# B&R Automation Studio project BaseProject (part 4)

#### Cyclic.st - Init, cyclic, exit code
```iecst
PROGRAM _CYCLIC

	MC_BR_SegCommandError_AcpTrak_0(Segment := ADR(TrackDiag.Seg.SegList[0].McType));

	IF MC_BR_SegCommandError_AcpTrak_0.Done THEN
		MC_BR_SegCommandError_AcpTrak_0.Execute := FALSE;
	END_IF

	(***********************************ASSEMBLY INFORMATION******************************	)
	(*Read Assebly Status*)

	DiagFbs.Asm.ReadStatus.Enable	:= TRUE;
	DiagFbs.Asm.ReadStatus();

	IF DiagFbs.Asm.ReadStatus.Valid THEN
		TrackDiag.Asm.AssemblyDisabled 	:= DiagFbs.Asm.ReadStatus.AssemblyDisabled;
		TrackDiag.Asm.AssemblyErrorStop := DiagFbs.Asm.ReadStatus.AssemblyErrorStop;
		TrackDiag.Asm.AssemblyReady		:= DiagFbs.Asm.ReadStatus.AssemblyReady;
		TrackDiag.Asm.AssemblyHoming	:= DiagFbs.Asm.ReadStatus.AssemblyHoming;
		TrackDiag.Asm.AssemblyStopping	:= DiagFbs.Asm.ReadStatus.AssemblyStopping;
	END_IF

	(*Read Assembly Info *)

	DiagFbs.Asm.ReadInfo.Enable		:= TRUE;
	DiagFbs.Asm.ReadInfo();

	IF DiagFbs.Asm.ReadInfo.Valid THEN
		TrackDiag.Asm.CommunicationReady 	:= DiagFbs.Asm.ReadInfo.AssemblyInfo.CommunicationReady;
		TrackDiag.Asm.PowerOn				:= DiagFbs.Asm.ReadInfo.AssemblyInfo.PowerOn;
		TrackDiag.Asm.ReadyForPowerOn		:= DiagFbs.Asm.ReadInfo.AssemblyInfo.ReadyForPowerOn;
		TrackDiag.Asm.ShuttleInErrorStopCount := DiagFbs.Asm.ReadInfo.AssemblyInfo.ShuttlesInErrorStopCount;
		TrackDiag.Asm.StartupCount			:= DiagFbs.Asm.ReadInfo.AssemblyInfo.StartupCount;
	END_IF

	(****************************** SEGMENT ERROR INFORMATION *****************************************)

	FOR SegIndex := 0 TO NUM_SEG DO

		IF TrackDiag.Seg.SegList[SegIndex].McType.controlif <> 0 THEN //If the array contains a segment reference

			DiagFbs.Seg.ReadInfo[SegIndex].Segment 	:= ADR(TrackDiag.Seg.SegList[SegIndex].McType);
			DiagFbs.Seg.ReadInfo[SegIndex].Enable	:= TRUE;
			DiagFbs.Seg.ReadInfo[SegIndex]();

			IF DiagFbs.Seg.ReadInfo[SegIndex].Valid THEN
				//Capture Segment Info
				TrackDiag.Seg.SegList[SegIndex].Status.CommunicationReady 	:= DiagFbs.Seg.ReadInfo[SegIndex].SegmentInfo.CommunicationReady;
				TrackDiag.Seg.SegList[SegIndex].Status.ReadyForPowerOn		:= DiagFbs.Seg.ReadInfo[SegIndex].SegmentInfo.ReadyForPowerOn;
				TrackDiag.Seg.SegList[SegIndex].Status.PowerOn				:= DiagFbs.Seg.ReadInfo[SegIndex].SegmentInfo.PowerOn;
				TrackDiag.Seg.SegList[SegIndex].Status.StartupCount			:= DiagFbs.Seg.ReadInfo[SegIndex].SegmentInfo.StartupCount;
				TrackDiag.Seg.SegList[SegIndex].Status.CommunicationState	:= DiagFbs.Seg.ReadInfo[SegIndex].SegmentInfo.CommunicationState;

			END_IF

			DiagFbs.Seg.ReadStatus[SegIndex].Segment := ADR(TrackDiag.Seg.SegList[SegIndex].McType);
			DiagFbs.Seg.ReadStatus[SegIndex].Enable	:= TRUE;
			DiagFbs.Seg.ReadStatus[SegIndex]();

			IF DiagFbs.Seg.ReadStatus[SegIndex].Valid THEN

				//Check for change of state to ErrorStop to command reading error data, IF communication is ready
				IF ((TrackDiag.Seg.SegList[SegIndex].Status.SegmentErrorStop = FALSE AND DiagFbs.Seg.ReadStatus[SegIndex].SegmentErrorStop = TRUE))
					AND (TrackDiag.Seg.SegList[SegIndex].Status.CommunicationReady = TRUE) THEN

					SegErrorCheck[SegIndex].CmdCheckErrorCode := TRUE;

					//Check for change of state from ErrorStop to reset error number in diag structure
				ELSIF ((TrackDiag.Seg.SegList[SegIndex].Status.SegmentErrorStop = TRUE) AND (DiagFbs.Seg.ReadStatus[SegIndex].SegmentErrorStop = FALSE))
					AND (TrackDiag.Seg.SegList[SegIndex].Status.CommunicationReady = TRUE) THEN

					TrackDiag.Seg.SegList[SegIndex].Status.ErrorCode := 0;

				END_IF
				//Capture Segment Status

				TrackDiag.Seg.SegList[SegIndex].Status.SegmentDisabled	:= DiagFbs.Seg.ReadStatus[SegIndex].SegmentDisabled;
				TrackDiag.Seg.SegList[SegIndex].Status.SegmentErrorStop	:= DiagFbs.Seg.ReadStatus[SegIndex].SegmentErrorStop;
				TrackDiag.Seg.SegList[SegIndex].Status.SegmentReady		:= DiagFbs.Seg.ReadStatus[SegIndex].SegmentReady;
				TrackDiag.Seg.SegList[SegIndex].Status.SegmentStopping	:= DiagFbs.Seg.ReadStatus[SegIndex].SegmentStopping;
			END_IF
		END_IF
	END_FOR

	CpuSim := DiagCpuIsSimulated() OR DiagCpuIsARsim();

	IF CpuSim = FALSE THEN
		actCheckErrorCode;
	END_IF

	(***********************************TRACKMAP******************************)

	paperCore();

	// compare the elementID clicked on in paper with the configured ID to find and set the array index for the list binding
	FOR SegIndex:= 0 TO NUM_SEG DO

		// clickId contains a leading # which needs to be removed,
		// the second compare checks against the text and arrow and deletes the first two letters because the SVG elements text and arrow have an added x leading the name
		IF TrackDiag.Seg.SegList[SegIndex].Name = DELETE(clickId,1,1) OR TrackDiag.Seg.SegList[SegIndex].Name = DELETE(clickId,2,1)THEN
			clickedSegment := TrackDiag.Seg.SegList[SegIndex];
			EXIT;
		END_IF
	END_FOR
END_PROGRAM
```

#### Types.typ - Local data types
```iecst
TYPE
	CheckStateEnum :
		(
		WAIT_FOR_CHECK,
		READ_DATA,
		READ_DATA_SEG_STATE,
		CHECK_SEG_STATE,
		READ_DATA_SEG_ERROR_STAT,
		CHECK_ERROR_STAT,
		READ_DATA_SEG_ERROR,
		CHECK_ERROR_CODE,
		WRITE_WARNING_CODE,
		READ_DATA_SEG_LAG,
		CHECK_SEG_LAG,
		READ_DATA_SEG_VEL,
		CHECK_SEG_VEL,
		READ_DATA_SEG_TEMP,
		CHECK_DATA_SEG_TEMP,
		WRITE_SPEED_FILTER,
		WRITE_SPEED_FILTER_WAIT,
		WRITE_ZERO_PITCH,
		READ_EXEC_ERROR,
		READ_SEG_STATUS,
		WRITE_SEG_RESET,
		WAIT_FOR_DONE
		);
	SegErrorCheckType : 	STRUCT
		CheckState : CheckStateEnum;
		CmdCheckErrorCode : BOOL;
		DataReadExecutionError : BOOL;
		ErrorNumber : UINT;
		SegStatusBits : UDINT;
		ErrorStatusBit : BOOL;
		ErrorStatus : UDINT;
	END_STRUCT;
	SegShuttleMonitorType : 	STRUCT
		CheckState_enum : BOOL;
		CmdMonitorLag : BOOL;
		CmdMonitorVelocity : BOOL;
		Lag : ARRAY[0..2]OF LREAL;
		Velocity : ARRAY[0..2]OF LREAL;
		LagLimitExceeded : BOOL;
		VelLimitExceeded : BOOL;
	END_STRUCT;
END_TYPE
```

#### Variables.var - Local variables
```iecst
VAR
	SegIndex : USINT;
	ErrorCodeIDInfo : ARRAY[0..NUM_SEG] OF McAcpTrakSegProcessParIDType;
	SegWarningCmdIDInfo : McAcpTrakSegProcessParIDType;
	SegErrorCheck : ARRAY[0..NUM_SEG] OF SegErrorCheckType;
	CpuSim : BOOL;
END_VAR
(*For testing only*)
VAR
	MC_BR_SegCommandError_AcpTrak_0 : MC_BR_SegCommandError_AcpTrak;
END_VAR
(*Declarations for TrackMap*)
VAR
	paperCore : TrkPaperCore;
	paperOptions : TrkPaperCoreOptionsType;
	clickId : STRING[160];
	clickedSegment : TrkDiagSegmentType;
	TrackDiag : TrkDiagStatusType;
	DiagFbs : DiagFbsType;
END_VAR
```

#### CheckErrorCode.st
```iecst
ACTION actCheckErrorCode:

	FOR SegIndex := 0 TO NUM_SEG DO

		CASE SegErrorCheck[SegIndex].CheckState OF

			WAIT_FOR_CHECK:
				//Wait for the command to check the error code ParID on the segment
				DiagFbs.Seg.ProcessParID[SegIndex].Execute := FALSE;

				IF SegErrorCheck[SegIndex].CmdCheckErrorCode THEN
					DiagFbs.Seg.ProcessParID[SegIndex].Execute := TRUE;
					DiagFbs.Seg.ProcessParID[SegIndex].Mode := mcACPTRAK_SEG_PARID_GET_NO_NCT;
					DiagFbs.Seg.ProcessParID[SegIndex].DataAddress := ADR(ErrorCodeIDInfo[SegIndex]);
					SegErrorCheck[SegIndex].CheckState := READ_DATA_SEG_ERROR;
					SegErrorCheck[SegIndex].CmdCheckErrorCode := FALSE; //Reset check command

				END_IF

			READ_DATA_SEG_ERROR:
				//Check for completion of reading the PARID for

				IF DiagFbs.Seg.ProcessParID[SegIndex].Done THEN
					//If the parID was successfully read, go to check error code state
					SegErrorCheck[SegIndex].CheckState := CHECK_ERROR_CODE;
					DiagFbs.Seg.ProcessParID[SegIndex].Execute := FALSE;
					SegErrorCheck[SegIndex].DataReadExecutionError := FALSE;

				ELSIF DiagFbs.Seg.ProcessParID[SegIndex].Error THEN
					//If there was an error in reading, go to error start
					SegErrorCheck[SegIndex].CheckState := READ_EXEC_ERROR;
				END_IF
			CHECK_ERROR_CODE:

				IF (SegErrorCheck[SegIndex].ErrorNumber = 0) OR (SegErrorCheck[SegIndex].ErrorNumber = 36005) THEN
					//Segment has no new error recorded. Shows either 0 or the commanded warning (36005) used to overwrite old errors
					TrackDiag.Seg.SegList[SegIndex].Status.ErrorCode := 0;
					SegErrorCheck[SegIndex].CheckState := WAIT_FOR_CHECK;
					TrackDiag.Seg.SegList[SegIndex].Status.Error := FALSE;

				ELSE
					//Otherwise, there is a new error on this segment
					TrackDiag.Seg.SegList[SegIndex].Status.ErrorCode := SegErrorCheck[SegIndex].ErrorNumber;

					TrackDiag.Seg.SegList[SegIndex].Status.Error := TRUE;
					//Send to overwrite state to store a known error number (36005) in the error code parID
					SegErrorCheck[SegIndex].CheckState := WRITE_WARNING_CODE;

				END_IF
			WRITE_WARNING_CODE:
				//Write commanded warning code (36005) to error parid
				DiagFbs.Seg.ProcessParID[SegIndex].DataAddress := ADR(SegWarningCmdIDInfo);
				DiagFbs.Seg.ProcessParID[SegIndex].ChannelIndex := 0;
				DiagFbs.Seg.ProcessParID[SegIndex].Mode := mcACPTRAK_SEG_PARID_SET;
				DiagFbs.Seg.ProcessParID[SegIndex].NumberOfParIDs := 0;
				DiagFbs.Seg.ProcessParID[SegIndex].Execute := TRUE;

				IF DiagFbs.Seg.ProcessParID[SegIndex].Done THEN
					//return to wait state
					DiagFbs.Seg.ProcessParID[SegIndex].Execute := FALSE;
					SegErrorCheck[SegIndex].CheckState := WAIT_FOR_CHECK;

				ELSIF DiagFbs.Seg.ProcessParID[SegIndex].Error THEN
					SegErrorCheck[SegIndex].CheckState := READ_EXEC_ERROR;
				END_IF
			READ_EXEC_ERROR:
				DiagFbs.Seg.ProcessParID[SegIndex].Execute := FALSE;
				SegErrorCheck[SegIndex].DataReadExecutionError := TRUE;

				IF DiagFbs.Seg.ProcessParID[SegIndex].Error = FALSE THEN
					SegErrorCheck[SegIndex].CheckState := WAIT_FOR_CHECK;
				END_IF
		END_CASE
	DiagFbs.Seg.ProcessParID[SegIndex]();
	END_FOR
END_ACTION
```

#### SegDefinition.st - not listed in the package file held
```iecst
//This file was automatically generated using the TrakMapImporter program. Verify that the segment names and assembly name match your project values correctly
ACTION SegDefinition:
	TrackDiag.Seg.SegList[0].Name  := 'gSeg_A_1';		TrackDiag.Seg.SegList[0].McType := gSeg_A_1;
	TrackDiag.Seg.SegList[1].Name  := 'gSeg_A_2';		TrackDiag.Seg.SegList[1].McType := gSeg_A_2;
	TrackDiag.Seg.SegList[2].Name  := 'gSeg_A_3';		TrackDiag.Seg.SegList[2].McType := gSeg_A_3;
	TrackDiag.Seg.SegList[3].Name  := 'gSeg_A_4';		TrackDiag.Seg.SegList[3].McType := gSeg_A_4;
	TrackDiag.Seg.SegList[4].Name  := 'gSeg_A_5';		TrackDiag.Seg.SegList[4].McType := gSeg_A_5;
	TrackDiag.Seg.SegList[5].Name  := 'gSeg_A_6';		TrackDiag.Seg.SegList[5].McType := gSeg_A_6;
	TrackDiag.Seg.SegList[6].Name  := 'gSeg_A_7';		TrackDiag.Seg.SegList[6].McType := gSeg_A_7;
	TrackDiag.Seg.SegList[7].Name  := 'gSeg_A_8';		TrackDiag.Seg.SegList[7].McType := gSeg_A_8;
	TrackDiag.Seg.SegList[8].Name  := 'gSeg_A_9';		TrackDiag.Seg.SegList[8].McType := gSeg_A_9;
	TrackDiag.Seg.SegList[9].Name  := 'gSeg_A_10';		TrackDiag.Seg.SegList[9].McType := gSeg_A_10;
	TrackDiag.Seg.SegList[10].Name  := 'gSeg_A_11';		TrackDiag.Seg.SegList[10].McType := gSeg_A_11;
	TrackDiag.Seg.SegList[11].Name  := 'gSeg_A_12';		TrackDiag.Seg.SegList[11].McType := gSeg_A_12;

	TrackDiag.Seg.SegCount := 12;

	TrackDiag.Seg.SegListAdr := ADR(TrackDiag.Seg.SegList);

	DiagFbs.Asm.ReadInfo.Assembly := ADR(DiagInterface.SampleTrak);
	DiagFbs.Asm.ReadStatus.Assembly := ADR(DiagInterface.SampleTrak);
END_ACTION
```

### Package Logical/Source/Assembly - EquipmentModule1

### Program Logical/Source/Assembly/AsmAlarm

#### Variables.var
```iecst
VAR
	fbAlarmTrakModule : MpAlarmXCore;
	FilterConfiguration : STRING[1000] := '';
	SortConfiguration : STRING[1000] := '';
	HistoryFilter : STRING[2000] := '';
	HistorySort : STRING[2000] := '';
	TriggerTestAlarm : BOOL;
	TriggerTestWarning : BOOL;
	TriggerTestInformation : BOOL;
END_VAR
```

#### Main.st
```iecst
PROGRAM _INIT
	(* Insert code here *)
	FilterConfiguration;
	SortConfiguration;
	HistoryFilter;
	HistorySort;
	gAlarmXCore_TrakModule;

END_PROGRAM

PROGRAM _CYCLIC
	(* Insert code here *)

	fbAlarmTrakModule(MpLink := ADR(TrakInterface.AlarmCore), Enable := TRUE);

	TriggerTestAlarm;
	TriggerTestInformation;
	TriggerTestWarning;

END_PROGRAM

PROGRAM _EXIT
	(* Insert code here *)

END_PROGRAM
```

### Program Logical/Source/Assembly/AsmConfig

#### Main.st
```iecst
PROGRAM _INIT
	(* Insert code here *)
	ModuleName := 'TrakModule';

END_PROGRAM

PROGRAM _CYCLIC
	(* Insert code here *)

END_PROGRAM

PROGRAM _EXIT
	(* Insert code here *)

END_PROGRAM
```

### Program Logical/Source/Assembly/AsmSampleTrak

#### Variables.var
```iecst
VAR
	fbSecAddShuttle : MC_BR_SecAddShuttle_AcpTrak;
	AssemblyState : TrBaseAsmStateEnum;
	fbAsmReadStatus : MC_BR_AsmReadStatus_AcpTrak;
	fbAsmReadInfo : MC_BR_AsmReadInfo_AcpTrak;
	fbAsmPowerOn : MC_BR_AsmPowerOn_AcpTrak;
	fbAsmPowerOff : MC_BR_AsmPowerOff_AcpTrak;
	fbAsmReset : MC_BR_AsmReset_AcpTrak;
	fbTrakModule : MpPackMLModule;
	parTrakModule : MpPackMLModuleParType;
END_VAR
```

#### Main.st
```iecst
(*******************************************************************************
 * Copyright: B&R Industrial Automation
 * Author:    Tyler Matijevich
 * Created:   November 5, 2020/12:35
********************************************************************************
 * Description: Control program to handle assembly power commands and error
 statuses
********************************************************************************)

PROGRAM _INIT
	fbSecAddShuttle.Sector := ADR(TrakInterface.SectorTrakA);
	fbSecAddShuttle.Position := 1000;

END_PROGRAM

PROGRAM _CYCLIC

	fbTrakModule(MpLink := ADR(TrakInterface.ModulePml),
					Enable := TRUE,
					Parameters := ADR(parTrakModule));

	// Reset command if no error
	IF gTrakSystem.Asm.Status.Error = FALSE THEN
		gTrakSystem.Asm.Cmd.ErrorReset := FALSE; // Force this command to reset
	END_IF

	(****************************************************************************************************
	****************************************************************************************************)
	(*
		Interrupts:
		1. Error status
		2. Stop command
		3. Read error
		4. ErrorStop state
	*)

	// 1. Skip remaining interrupt checks when an error exists
	IF gTrakSystem.Asm.Status.Error OR ShInit.Status.Error THEN
		// Go to ERROR
		AssemblyState := ASM_STATE_ERROR;

	// 2. Accept stop command
	ELSIF EDGENEG(gTrakSystem.Asm.Cmd.Power) THEN
		// Power off if powering or powered on
		IF gTrakSystem.Asm.Status.Homing OR gTrakSystem.Asm.Status.Ready THEN
			// Execute the power off command. Execute should not be true in either of these states
			fbAsmPowerOff.Execute := TRUE;
		END_IF

		// Go to OFF
		AssemblyState := ASM_STATE_OFF;

	// 3. The assembly read function blocks are in error
	ELSIF fbAsmReadStatus.Error OR fbAsmReadInfo.Error THEN
		// Log event
		// Set error status and go to ERROR
		gTrakSystem.Asm.Status.Error	:= TRUE;
		AssemblyState 				:= ASM_STATE_ERROR;

	// 4. Assembly in ErrorStop
	ELSIF gTrakSystem.Asm.Status.ErrorStop AND fbAsmReset.Busy = FALSE THEN
		// Log event
		// Set error status and go to ERROR
		gTrakSystem.Asm.Status.Error	:= TRUE;
		AssemblyState 				:= ASM_STATE_ERROR;

	END_IF

	(****************************************************************************************************
	****************************************************************************************************)
	// Main assembly state machine
	CASE AssemblyState OF
		// ----------------------------------------------------------------------------------------------------
		// OFF
		ASM_STATE_OFF:
			// Accept AsmPowerOff command
			IF fbAsmPowerOff.Done THEN
				// Reset execution
				fbAsmPowerOff.Execute := FALSE;

			ELSIF fbAsmPowerOff.Error THEN
				// Log event
				// Set error status and go to ERROR
				gTrakSystem.Asm.Status.Error	:= TRUE;
				AssemblyState 				:= ASM_STATE_ERROR;

			// Accept AsmReset command
			ELSIF fbAsmReset.Done THEN
				// Reset execution
				fbAsmReset.Execute := FALSE;

			ELSIF fbAsmReset.Error THEN
				// Log event
				// Set error status and go to ERROR
				gTrakSystem.Asm.Status.Error	:= TRUE;
				AssemblyState 				:= ASM_STATE_ERROR;

			// Wait for power command and assembly conditions
			ELSIF gTrakSystem.Asm.Cmd.Power AND gTrakSystem.Asm.Cmd.Stop = FALSE // Read input commands
			  AND gTrakSystem.Asm.Status.Disabled AND gTrakSystem.Asm.Status.ReadyForPowerOn // Check assembly statuses
			  AND fbAsmPowerOff.Execute = FALSE AND fbAsmReset.Execute = FALSE
			  (*AND MpPackMLStateIsActive(TrakInterface.ModulePml,mpPACKML_STATE_EXECUTE,1)*)
			  	THEN // Check other function block execution
				// Power on the assembly
				fbAsmPowerOn.Execute := TRUE;

				// Go to POWER
				AssemblyState := ASM_STATE_POWER;

			END_IF

		// ----------------------------------------------------------------------------------------------------
		// POWER
		ASM_STATE_POWER:
			// Wait for the power on command to complete, ensure correct statuses
			IF fbAsmPowerOn.Done AND gTrakSystem.Asm.Status.Ready AND gTrakSystem.Asm.Status.PowerOn THEN
				// Reset execution
				fbAsmPowerOn.Execute := FALSE;

				// Go to READY
				AssemblyState := ASM_STATE_READY;

//				// Check shuttle initialization for ready status
//				IF ShInit.Status.Ready THEN
//					// Start the shuttle initialization
//					ShInit.Cmd.Start := TRUE;
//
//					// Go to INIT
//					AssemblyState := ASM_STATE_INIT;
//
//				ELSE
//					// Log event
//					// Set error status and go to ERROR
//					gTrakSystem.Asm.Status.Error	:= TRUE;
//					AssemblyState 				:= ASM_STATE_ERROR;
//
//				END_IF

			ELSIF fbAsmPowerOn.Error THEN
				// Log event
				// Set error status and go to ERROR
				gTrakSystem.Asm.Status.Error	:= TRUE;
				AssemblyState 				:= ASM_STATE_ERROR;

			// Check if the assembly suddenly loses power
			ELSIF (gTrakSystem.Asm.Status.Disabled OR gTrakSystem.Asm.Status.PowerOn = FALSE)
			  AND fbAsmPowerOn.Execute = FALSE THEN
				// Log event
				// Set error status and go to ERROR
				gTrakSystem.Asm.Status.Error	:= TRUE;
				AssemblyState 				:= ASM_STATE_ERROR;

			END_IF

		// ----------------------------------------------------------------------------------------------------
		// INIT
		ASM_STATE_INIT:
		// Go to READY
				AssemblyState := ASM_STATE_READY;

			// Wait for the shuttle initialization to complete
//			IF ShInit.Status.Complete THEN
//				// Reset command
//				ShInit.Cmd.Start := FALSE;
//
//				// Go to READY
//				AssemblyState := ASM_STATE_READY;
//
//			ELSIF ShInit.Status.Error THEN
//				// Log event
//				// Set error status and go to ERROR
//				gTrakSystem.Asm.Status.Error	:= TRUE;
//				AssemblyState 				:= ASM_STATE_ERROR;
//
//			END_IF

		// ----------------------------------------------------------------------------------------------------
		// READY
		ASM_STATE_READY:
			// Check if the assembly suddenly becomes disabled
			IF gTrakSystem.Asm.Status.Disabled THEN
				// Log event
				// Set error status and go to ERROR
				gTrakSystem.Asm.Status.Error	:= TRUE;
				AssemblyState 				:= ASM_STATE_ERROR;

			END_IF

		// ----------------------------------------------------------------------------------------------------
		// ERROR
		ASM_STATE_ERROR:
			// Wait for an error reset command
			IF gTrakSystem.Asm.Cmd.ErrorReset THEN
				// If ErrorStop, reset the assembly
				IF gTrakSystem.Asm.Status.ErrorStop AND fbAsmReset.Error = FALSE THEN
					// Execute an assembly reset
					fbAsmReset.Execute := TRUE;

					// Reset other function block's execution
					fbAsmPowerOn.Execute 	:= FALSE;
					fbAsmPowerOff.Execute	:= FALSE;

				// If powered
				ELSIF (gTrakSystem.Asm.Status.Homing OR gTrakSystem.Asm.Status.Ready) AND fbAsmPowerOff.Error = FALSE THEN
					// Power off the assembly
					fbAsmPowerOff.Execute := TRUE;

					// Reset other function block's execution
					fbAsmPowerOn.Execute 	:= FALSE;
					fbAsmReset.Execute		:= FALSE;

				ELSE
					// Reset all function block's execution
					fbAsmPowerOn.Execute 	:= FALSE;
					fbAsmPowerOff.Execute	:= FALSE;
					fbAsmReset.Execute		:= FALSE;

				END_IF // Check assembly state

				// Reset the error bit and go back to OFF
				gTrakSystem.Asm.Status.Error	:= FALSE;
				AssemblyState				:= ASM_STATE_OFF;

			END_IF

	END_CASE // Assembly state machine

	// Call all mapp Trak function blocks
	fbAsmReadStatus(Assembly := ADR(gSampleTrak), Enable := TRUE); // Always enable to reduce logger entries
	fbAsmReadInfo(Assembly := ADR(gSampleTrak), Enable := TRUE); // Always enable to reduce logger entries
	fbAsmPowerOn(Assembly := ADR(gSampleTrak));
	fbAsmPowerOff(Assembly := ADR(gSampleTrak));
	fbAsmReset(Assembly := ADR(gSampleTrak));
	fbSecAddShuttle();
	fbSecAddShuttle.Execute := FALSE;

	// Update the global status information
	gTrakSystem.Asm.Status.Disabled					:= fbAsmReadStatus.Valid AND fbAsmReadStatus.AssemblyDisabled;
	gTrakSystem.Asm.Status.Homing					:= fbAsmReadStatus.Valid AND fbAsmReadStatus.AssemblyHoming;
	gTrakSystem.Asm.Status.Ready					:= fbAsmReadStatus.Valid AND fbAsmReadStatus.AssemblyReady;
	gTrakSystem.Asm.Status.Stopping					:= fbAsmReadStatus.Valid AND fbAsmReadStatus.AssemblyStopping;
	gTrakSystem.Asm.Status.ErrorStop				:= fbAsmReadStatus.Valid AND fbAsmReadStatus.AssemblyErrorStop;
	gTrakSystem.Asm.Status.CommunicationReady		:= fbAsmReadInfo.Valid AND fbAsmReadInfo.AssemblyInfo.CommunicationReady;
	gTrakSystem.Asm.Status.ReadyForPowerOn			:= fbAsmReadInfo.Valid AND fbAsmReadInfo.AssemblyInfo.ReadyForPowerOn;
	gTrakSystem.Asm.Status.PowerOn					:= fbAsmReadInfo.Valid AND fbAsmReadInfo.AssemblyInfo.PowerOn;
	gTrakSystem.Asm.Status.ShuttlesInErrorStopCount	:= fbAsmReadInfo.AssemblyInfo.ShuttlesInErrorStopCount; // If not valid, assuming these are zero
	gTrakSystem.Asm.Status.StartupCount				:= fbAsmReadInfo.AssemblyInfo.StartupCount;

	// Call all subroutine actions
	ShInit.Cmd.Stop := gTrakSystem.Asm.Status.Ready = FALSE;
//	ShuttleInitialization;

END_PROGRAM

PROGRAM _EXIT

END_PROGRAM
```

### SM11.var
```iecst
(*Shuttle initialization variables*)
VAR
	colorIndex : UDINT;
	BufferReturnIndex : TrBaseErrorCodeEnum;
	fbAsmGetShuttle : MC_BR_AsmGetShuttle_AcpTrak;
	fbShCopyUserData : MC_BR_ShCopyUserData_AcpTrak;
	fbRoutedMoveVel_AcpTrak : MC_BR_RoutedMoveVel_AcpTrak;
END_VAR
```

### Program Logical/Source/Assembly/SubModule1/ShuttleInit

#### Main.st
```iecst
PROGRAM _INIT
	(* Insert code here *)
	 TrakInterface;
END_PROGRAM

PROGRAM _CYCLIC
	// Reset status variables, they will be set in the respective state
	ShInit.Status.Ready 	:= FALSE;
	ShInit.Status.Complete	:= FALSE;

	(*
		Interrupts:
		1. Error status
		2. Stop command
	*)
	// 1. Check error status
	IF ShInit.Status.Error THEN
		// Go to ERROR, skip remaining interrupts
		ShInitState := 255;

	// 2. Accept stop commands
	ELSIF ShInit.Cmd.Stop THEN
		// Reset FB execution
		fbAsmGetShuttle.Enable		:= FALSE;
		fbShCopyUserData.Execute 	:= FALSE;

		// Go to INIT
		ShInitState := 0;

	END_IF

	// Shuttle initialization main state machine
	CASE ShInitState OF
		// ----------------------------------------------------------------------------------------------------
		// INIT
		0:
			// Set the status
			ShInit.Status.Ready := TRUE;

			// Wait to start
			IF (ShInit.Cmd.Start OR ShInit.Cmd.Cycle) AND ShInit.Cmd.Stop = FALSE THEN
				// Clear the shuttle buffer
				BufferReturnIndex := TrBaseClearShBuffer(ADR(gTrakSystem.Buffer), SIZEOF(gTrakSystem.Buffer));
				IF BufferReturnIndex = trBASE_NO_ERROR THEN
					// Enable the assembly get shuttle function block
					fbAsmGetShuttle.Assembly 	:= ADR(TrakInterface.SampleTrak);
					fbAsmGetShuttle.Enable 		:= TRUE;

					// Go to READ
					ShInitState := 10;

				ELSE
					// Log event
					// Set error status and go to ERROR
					ShInit.Status.Error := TRUE;
					ShInitState 		:= 255;

				END_IF
			END_IF // Start

		// ----------------------------------------------------------------------------------------------------
		// READ
		10:
			// Wait for a valid read, then read the shuttle
			IF fbAsmGetShuttle.Valid AND fbAsmGetShuttle.TotalCount > 0 THEN
				// Add the shuttle to the buffer
				BufferReturnIndex := TrBaseAddShToBuffer(fbAsmGetShuttle.Axis, ADR(gTrakSystem.Buffer), SIZEOF(gTrakSystem.Buffer));
				IF BufferReturnIndex = trBASE_NO_ERROR THEN
					// Shuttle added successfully, read the shuttle user data
					fbShCopyUserData.Axis 			:= ADR(fbAsmGetShuttle.Axis);
					fbShCopyUserData.DataAddress	:= ADR(ShuttleUserData);
					fbShCopyUserData.DataSize		:= SIZEOF(ShuttleUserData);
					fbShCopyUserData.Mode			:= mcACPTRAK_USERDATA_GET;
					fbShCopyUserData.Execute		:= TRUE;

					// Go to DATA
					ShInitState := 20;

				ELSE
					// Log event
					// Set error status and go to ERROR
					ShInit.Status.Error := TRUE;
					ShInitState 		:= 255;

				END_IF

			ELSIF fbAsmGetShuttle.Valid AND fbAsmGetShuttle.TotalCount = 0 THEN // No shuttles on the assembly
				// Go straight to the complete state
				ShInitState := 60;

			ELSIF fbAsmGetShuttle.Error THEN
				// Log event
				// Set error status and go to ERROR
				ShInit.Status.Error := TRUE;
				ShInitState 		:= 255;

			END_IF

		// ----------------------------------------------------------------------------------------------------
		// DATA
		20:
			IF fbShCopyUserData.Done THEN
				// Reset the command
				fbShCopyUserData.Execute := FALSE;

				// Go to WRITE
				ShInitState := 30;

			ELSIF fbShCopyUserData.Error THEN
				// Log event
				// Set error status and go to ERROR
				ShInit.Status.Error := TRUE;
				ShInitState 		:= 255;

			END_IF

		// ----------------------------------------------------------------------------------------------------
		// WRITE
		30:
			IF fbShCopyUserData.Done THEN
				// Shuttle user data write complete, shuttle ID set, reset the execution
				fbShCopyUserData.Execute := FALSE;

				// Reset the assembly get shuttle next command
				fbAsmGetShuttle.Next := FALSE;

				// Go to MOVE
				ShInitState := 35;

			ELSIF fbShCopyUserData.Error THEN
				// Log event
				// Set error status and go to ERROR
				ShInit.Status.Error := TRUE;
				ShInitState 		:= 255;

			ELSE
				// Execute the write command
				fbShCopyUserData.Mode		:= mcACPTRAK_USERDATA_SET;
				fbShCopyUserData.Execute 	:= TRUE;

				// Set the shuttle ID (if not already set)
				ShuttleUserData.ID := fbAsmGetShuttle.AdditionalInfo.ShuttleID;
				ShuttleUserData.Color := (colorIndex / 200) MOD 10;
				colorIndex := colorIndex + 1;

			END_IF

		// ----------------------------------------------------------------------------------------------------
		// MOVE
		35:
			fbRoutedMoveVel_AcpTrak.Axis			:= ADR(fbAsmGetShuttle.Axis);
			fbRoutedMoveVel_AcpTrak.Execute			:= TRUE;
			fbRoutedMoveVel_AcpTrak.Sector			:= ADR(TrakInterface.SectorTrakAll);
			fbRoutedMoveVel_AcpTrak.Position		:= 1;
			fbRoutedMoveVel_AcpTrak.Acceleration	:= 10.0;
			fbRoutedMoveVel_AcpTrak.Deceleration	:= 10.0;
			fbRoutedMoveVel_AcpTrak.Jerk			:= 0.0;
			fbRoutedMoveVel_AcpTrak.BufferMode		:= mcABORTING;
			fbRoutedMoveVel_AcpTrak.RouteVelocity	:= 1;
			fbRoutedMoveVel_AcpTrak.Velocity		:= 1;
			fbRoutedMoveVel_AcpTrak.AdvancedParameters.StartDirection := mcDIR_UNDEFINED;
			fbRoutedMoveVel_AcpTrak.AdvancedParameters.ShuttleOrientation := mcDIR_UNDEFINED;
			fbRoutedMoveVel_AcpTrak.AdvancedParameters.EndDirection := mcDIR_NEGATIVE;
			ShInitState := 40;

		// ----------------------------------------------------------------------------------------------------
		// UPDATE
		40:
			// Check for the next shuttle
			IF fbAsmGetShuttle.Valid AND fbAsmGetShuttle.RemainingCount > 0 THEN
				// Issue next command and go back to the READ state
				fbAsmGetShuttle.Next 	:= TRUE;
				ShInitState				:= 10;

			// Check when no shuttles remain
			ELSIF fbAsmGetShuttle.Valid AND fbAsmGetShuttle.RemainingCount = 0 THEN
				// All shuttles have been captured, reset the FB
				fbAsmGetShuttle.Enable := FALSE;

				// Go to DELETE
				ShInitState := 50;

			ELSIF fbAsmGetShuttle.Error THEN
				// Log event
				// Set error status and go to ERROR
				ShInit.Status.Error := TRUE;
				ShInitState 		:= 255;

			END_IF

		// ----------------------------------------------------------------------------------------------------
		// DELETE
		50:
			// Shuttle detection complete, now delete marked shuttles
			gTrakSystem.Tracking.Cmd.Delete := gTrakSystem.Tracking.Status.ShuttlesToBeDeletedCount <> 0;

			// Leave when no shuttles need to be deleted
			IF gTrakSystem.Tracking.Status.ShuttlesToBeDeletedCount = 0 THEN
				// Go to COMPLETE
				ShInitState := 60;
			END_IF

		// ----------------------------------------------------------------------------------------------------
		// COMPLETE
		60:
			// Set the status
			ShInit.Status.Complete := TRUE;

			// Return to INIT when the state command is reset
			IF ShInit.Cmd.Start = FALSE OR ShInit.Cmd.Cycle THEN
				// Go to INIT
				ShInitState := 0;
			END_IF

		// ----------------------------------------------------------------------------------------------------
		// ERROR
		255:
			// Wait for error reset command
			IF ShInit.Cmd.ErrorReset THEN
				// Reset the function blocks
				fbAsmGetShuttle.Enable 		:= FALSE;
				fbShCopyUserData.Execute 	:= FALSE;

				// Reset the error bit and go to INIT
				ShInit.Status.Error := FALSE;
				ShInitState 		:= 0;

			END_IF

	END_CASE

	// Call mapp Trak function blocks
	fbAsmGetShuttle();
	fbShCopyUserData();
	fbShCopyUserData();
	fbRoutedMoveVel_AcpTrak();
	fbRoutedMoveVel_AcpTrak.Execute := FALSE;

END_PROGRAM

PROGRAM _EXIT
	(* Insert code here *)

END_PROGRAM
```

### EMx.var
```iecst
VAR
	ModuleLink : STRING[40];
	ModuleName : STRING[40];
	ModuleInterface : ModuleInterfaceType;
END_VAR
(*Alarm configuration*)
VAR
	fbAlarmModule : MpAlarmXCore;
	ProcessAlarm : BOOL;
	ProcessWarning : BOOL;
	ProcessInformation : BOOL;
	fbModuleConfig : MpRecipeXml;
	ConfigCategory : STRING[50];
	ConfigHeader : MpRecipeXmlHeaderType;
	fbConfigRegPar : MpRecipeRegPar;
END_VAR
```

### Program Logical/Source/EMx/Config (IEC)

#### Main.st
```iecst
PROGRAM _INIT
	(* Insert code here *)

	ST_name(0,ADR(ModuleLink),0);

	IF (ModuleLink = 'EMx::ConfigEMx') THEN

		ModuleName := 'EMx';
		ConfigCategory := ModuleName;
		ConfigHeader.Version := '0.0.1';

	ELSIF (ModuleLink = 'EMx::ConfigEMx') THEN

		ModuleName := 'EMx';
		ConfigCategory := ModuleName;
		ConfigHeader.Version := '0.0.1';

	END_IF

	gPackMLModule_EMx;
	gRecipeXml_EMx;

END_PROGRAM

PROGRAM _CYCLIC
	(* Insert code here *)

	fbModuleConfig(MpLink := ADR(ModuleInterface.RecipeCore),
				Enable := TRUE,
				DeviceName := ADR('Config'),
				FileName := ADR(ModuleName),
				Header := ADR(ConfigHeader),
				Category := ADR(ConfigCategory));

	fbConfigRegPar(MpLink := ADR(ModuleInterface.RecipeCore), Enable := TRUE , PVName := ADR('ModuleInterface'), Category := ADR(ConfigCategory));

	ProcessInformation;
	ProcessWarning;
	ProcessAlarm;

END_PROGRAM

PROGRAM _EXIT
	(* Insert code here *)

END_PROGRAM
```

### Program Logical/Source/EMx/Alarm (IEC)

#### Main.st - Init, cyclic, exit code
```iecst
PROGRAM _INIT

	//call each variable for mappView
	FilterConfiguration;
	SortConfiguration;
	HistoryFilter;
	HistorySort;

	//call each AlarmX MpLink so it variable exists in memory and can be used in the AppModule variable mapping
	gAlarmXCore_EMx;

END_PROGRAM

PROGRAM _CYCLIC
	(* Call alarm core component *)

	fbAlarmModule(MpLink := ADR(ModuleInterface.AlarmCore), Enable := TRUE);

END_PROGRAM

PROGRAM _EXIT
	(* Insert code here *)

END_PROGRAM
```

#### Variables.var - Local variables
```iecst
VAR
	FilterConfiguration : STRING[1000] := '';
	SortConfiguration : STRING[1000] := '';
	HistoryFilter : STRING[2000] := '';
	HistorySort : STRING[2000] := '';
END_VAR
```

### Program Logical/Source/EMx/Process (IEC)

#### Variables.var
```iecst
VAR
	Counter : UDINT;
END_VAR
```

#### Main.st
```iecst
PROGRAM _INIT
	(* Insert code here *)

END_PROGRAM

PROGRAM _CYCLIC
	(* Insert code here *)

	IF MpPackMLStateIsActive(ModuleInterface.MainPml,mpPACKML_STATE_EXECUTE,1) THEN
		Counter := Counter + 1;
	END_IF

	ProcessAlarm;
	ProcessWarning;
	ProcessInformation;

END_PROGRAM

PROGRAM _EXIT
	(* Insert code here *)

END_PROGRAM
```

### Source.var
```iecst
VAR
	ModuleLink : STRING[40];
	ModuleName : STRING[40];
	StartValue : INT;
	Counter : INT;
	ModuleInterface : ModuleInterfaceType;
END_VAR
(*Alarm configuration*)
VAR
	fbAlarmModule : MpAlarmXCore;
	FilterConfiguration : STRING[1000] := '';
	SortConfiguration : STRING[1000] := '';
	HistoryFilter : STRING[2000] := '';
	HistorySort : STRING[2000] := '';
	ConfigAlarm : BOOL;
	ConfigWarning : BOOL;
	ConfigInformation : BOOL;
	RecoveryAlarm : BOOL;
	RecoveryWarning : BOOL;
	RecoveryInformation : BOOL;
	OperationAlarm : BOOL;
	OperationWarning : BOOL;
	OperationInformation : BOOL;
	fbModuleConfig : MpRecipeXml;
	ConfigCategory : STRING[50];
	ConfigHeader : MpRecipeXmlHeaderType;
	fbConfigRegPar : MpRecipeRegPar;
END_VAR
```

### Program Logical/Source/ReusableSource/Alarm (IEC)

#### Main.st
```iecst
PROGRAM _INIT

	//call each variable for mappView
	FilterConfiguration;
	SortConfiguration;
	HistoryFilter;
	HistorySort;

	//call each AlarmX MpLink so it variable exists in memory and can be used in the AppModule variable mapping
	gAlarmXCore_EM2;
	gAlarmXCore_EM3;

END_PROGRAM

PROGRAM _CYCLIC
	(* Call alarm core component *)

	fbAlarmModule(MpLink := ADR(ModuleInterface.AlarmCore), Enable := TRUE);

END_PROGRAM

PROGRAM _EXIT
	(* Insert code here *)

END_PROGRAM
```

### Program Logical/Source/ReusableSource/BarrierCtrl (IEC)

#### Main.st
```iecst
PROGRAM _INIT
	(* Insert code here *)

END_PROGRAM

PROGRAM _CYCLIC
	(* Insert code here *)

END_PROGRAM

PROGRAM _EXIT
	(* Insert code here *)

END_PROGRAM
```

### SampleTrak.typ
```iecst
(*==================================================
ACOPOStrak Global Structure Hierarchy
==================================================*)

TYPE
	TrakType : 	STRUCT  (*Global structure definition*)
		Asm : TrBaseAsmType; (*Assembly substructure*)
		Par : TrakParametersType; (*ACOPOStrak application parameters*)
		Buffer : ARRAY[0..149]OF BOOL;
		Tracking : TrBaseTrackingType;
	END_STRUCT;
END_TYPE

(*Application parameters*)

TYPE
	TrakParametersType : 	STRUCT
		Velocity : REAL;
		Acceleration : REAL;
		CriticalVelocity : REAL;
		RecoveryVelocity : REAL;
	END_STRUCT;
END_TYPE

(*Interface for variable mapping*)

TYPE
	ModuleInterfaceType : 	STRUCT
		SampleTrak : McAssemblyType;
		MainPml : MpComIdentType;
		ModulePml : MpComIdentType;
		AlarmCore : MpComIdentType;
		AuditCore : MpComIdentType;
		RecipeCore : MpComIdentType;
	END_STRUCT;
END_TYPE
```

### Program Logical/Source/SampleTrak/TSM (IEC)

#### Variables.var
```iecst
VAR
	fbMainTsm : MpPackMLModule;
	parMainTsm : MpPackMLModuleParType;
END_VAR
```

#### Main.st
```iecst
PROGRAM _INIT

END_PROGRAM

PROGRAM _CYCLIC
	(* Insert code here *)

	fbMainTsm(MpLink := ADR(gMainModule),
						Enable := TRUE,
						Parameters := ADR(parMainTsm));

	MpPackMLStateIsActive(gMainModule,mpPACKML_STATE_EXECUTE,1);

END_PROGRAM

PROGRAM _EXIT
	(* Insert code here *)

END_PROGRAM
```

- Program Logical/Source/SampleTrak/TSMMain (IEC) (no source held here)

### Program Logical/Source/SampleTrak/TSMAlarm (IEC)

#### Variables.var
```iecst
VAR
	fbAlarmMainTSM : MpAlarmXCore;
	FilterConfiguration : STRING[1000] := '';
	SortConfiguration : STRING[1000] := '';
	HistoryFilter : STRING[2000] := '';
	HistorySort : STRING[2000] := '';
	fbAlarmHistMainTSM : MpAlarmXHistory;
	TriggerTestAlarm : BOOL;
	MpAlarmXListUI_0 : MpAlarmXListUI;
	UIConnect : MpAlarmXListUIConnectType;
END_VAR
```

#### Main.st
```iecst
PROGRAM _INIT
	(* Insert code here *)
	FilterConfiguration;
	SortConfiguration;
	HistoryFilter;
	HistorySort;
END_PROGRAM

PROGRAM _CYCLIC
	(* Insert code here *)
	fbAlarmMainTSM(MpLink := ADR(gAlarmXCore), Enable := TRUE);
	fbAlarmHistMainTSM(MpLink := ADR(gAlarmXHistory), Enable := TRUE, DeviceName := ADR('User'));

	MpAlarmXListUI_0(MpLink := ADR(gAlarmXCore), Enable := TRUE,UIConnect := ADR(UIConnect));

	TriggerTestAlarm;

END_PROGRAM

PROGRAM _EXIT
	(* Insert code here *)

END_PROGRAM
```

### TrackDiagGlobal.typ
```iecst
(*Insert your comment here.*)

TYPE
	DiagStatusType : 	STRUCT
		Sys : SystemStatusType;
		Asm : AsmStatusType;
		Seg : SegmentDataType;
		Shuttle : ShuttleStatusType;
		PS : ARRAY[0..NUM_PS]OF PowerSupplyStatusType;
		Hub : ARRAY[0..NUM_HUBS]OF HubStatusType;
		IO : IOStatusType;
		CPU : CPUStatusType;
	END_STRUCT;
	SystemStatusType : 	STRUCT
		ConfigCheckComplete : BOOL;
		ConfigCheckOk : BOOL;
		StatusMessage : STRING[0];
	END_STRUCT;
	AsmStatusType : 	STRUCT
		AssemblyDisabled : BOOL;
		AssemblyReady : BOOL;
		AssemblyHoming : BOOL;
		AssemblyStopping : BOOL;
		AssemblyErrorStop : BOOL;
		CommunicationReady : BOOL;
		ReadyForPowerOn : BOOL;
		PowerOn : BOOL;
		StartupCount : UDINT;
		ShuttleInErrorStopCount : UINT;
	END_STRUCT;
	ShuttleStatusType : 	STRUCT
		Position : REAL;
		Velocity : REAL;
		LagError : REAL;
		Segment : REAL;
		Channel_ID : REAL;
		ErrorMessage : STRING[0];
	END_STRUCT;
	PowerSupplyStatusType : 	STRUCT
		ModuleOk : BOOL;
		CurrentLimit01 : BOOL;
		Voltage01 : SINT;
		Current01 : INT;
		ClearOutput01 : BOOL;
		ErrorOutput01 : BOOL;
		OverloadError01 : BOOL;
		StatusPhaseDetection01 : BOOL;
		StatusOvertemperture01 : BOOL;
		StatusOvervoltage01 : BOOL;
		ChopperActive01 : BOOL;
		StatusChopper01 : BOOL;
		StatusBleeder01 : BOOL;
		StatusOutput02 : BOOL;
	END_STRUCT;
	HubStatusType : 	STRUCT
		ErrorMessage : STRING[0];
		X20BC8083_ModuleOK : BOOL;
		X20PS9400_ModuleOk : BOOL;
		X20PS9400_StatusInput01 : BOOL;
		X20PS9400_StatusInput02 : BOOL;
		PLK_LinkOk : BOOL;
		PLK_CycleOk : BOOL;
		PLK_SyncOk : BOOL;
	END_STRUCT;
	IOStatusType : 	STRUCT
		X20BT9400_ModuleOk : BOOL;
		X20BT9400_StatusInput01 : BOOL;
		X20BT9400_StatusInput02 : BOOL;
		X20DI2371_ModuleOk : BOOL;
		X20DI2371_DigitalInput01 : BOOL;
		X20DI2371_DigitalInput02 : BOOL;
	END_STRUCT;
	CPUStatusType : 	STRUCT
		TemperatureCPU : UINT;
		TemperatureBoard : UINT;
	END_STRUCT;
	ErrorSegInfoType : 	STRUCT
		Error : USINT;
	END_STRUCT;
END_TYPE

(*LogBook def*)

TYPE
	LogBookStateEnum :
		( (*State machine*)
		STATE_WAIT,
		STATE_CREATE,
		STATE_OPEN,
		STATE_LATEST,
		STATE_NEXT,
		STATE_DETAILS_1,
		STATE_DETAILS_2,
		STATE_DETAILS_3,
		STATE_CHECK_FILTER,
		STATE_UPDATE_LIST,
		STATE_DETAILS_4,
		STATE_FILTER,
		STATE_PREP,
		STATE_ERROR,
		STATE_NONE
		);
	LogBookSeverityEnum :
		(
		SEVERITY_NOTIFICATION,
		SEVERITY_INFORMATION,
		SEVERITY_WARNING,
		SEVERITY_ERROR
		);
	LogBookTypeEnum :
		(
		LOG_ACCESS_SECURITY,
		LOG_COMMISIONING,
		LOG_CONNECTIVITY,
		LOG_FIELDBUS,
		LOG_FIREWALL,
		LOG_MAPP,
		LOG_MOTION,
		LOG_SAFETY,
		LOG_SYSTEM,
		LOG_TEXTSYSTEM,
		LOG_UNITSYSTEM,
		LOG_USER,
		LOG_VISUALIZATION
		);
	LogBookSortingEnum :
		(
		SORTING_ASC,
		SORTING_DESC
		);
	LogBookParType : 	STRUCT  (*Parameter structure*)
		DateNow : DATE_AND_TIME; (*Current date and time*)
		TableConfig : STRING[100]; (*Hide unused rows*)
		EntriesMax : UINT; (*Maximum number of entries, shadow of LOGBOOK_ENTRIES_MAX*)
		FilterErrorNo : UDINT; (*Filter by error number*)
		FilterErrorText : STRING[LOGBOOK_TEXT_LEN]; (*Filter by error text*)
		FilterSeverity : ARRAY[0..3]OF BOOL := [4(TRUE)]; (*Filter by severity*)
		FilterLogbook : ARRAY[0..LOGBOOK_BOOKS_MAX]OF BOOL := [14(TRUE)]; (*Filter by logbook*)
		FilterDateStart : DATE; (*Filter by date*)
		FilterDateEnd : DATE;
		Sorting : LogBookSortingEnum := SORTING_DESC; (*Sort date asc or desc*)
		AbortOnEntriesLimit : BOOL; (*Stop looking for additional entries when limit is reached*)
		AutoUpdate : BOOL; (*Automatically update data*)
		AutoUpdateInterval : UINT := 60; (*Interval for auto update in s*)
		CreateErrorNo : UINT; (*Error no for new entry*)
		CreateErrorText : STRING[LOGBOOK_TEXT_LEN]; (*Error text for new entry*)
		CreateSeverity : LogBookSeverityEnum := SEVERITY_NOTIFICATION; (*Error severiry for new entry*)
		CreateLogbook : LogBookTypeEnum := LOG_USER; (*Error logbook for new entry*)
	END_STRUCT;
	LogBookErrorType : 	STRUCT  (*Error structure*)
		State : LogBookStateEnum; (*State where the error occured*)
	END_STRUCT;
	LogBookDataType : 	STRUCT  (*Data structure*)
		Entries : LogBookDataEntryType;
		EntriesTotal : UINT; (*Total number of entries*)
		CntSeverity : ARRAY[0..3]OF UINT; (*Counts by severity*)
		CntLogbook : ARRAY[0..LOGBOOK_BOOKS_MAX]OF UINT; (*Counts by logbook*)
		LastUpdate : STRING[25]; (*Last refresh run*)
	END_STRUCT;
	LogBookDataEntryType : 	STRUCT  (*Entries structure*)
		EventID : ARRAY[1..LOGBOOK_ENTRIES_MAX]OF DINT; (*Event ID*)
		Timestamp : ARRAY[1..LOGBOOK_ENTRIES_MAX]OF STRING[25]; (*Date and time*)
		DTsec : ARRAY[1..LOGBOOK_ENTRIES_MAX]OF UDINT; (*Date and time in sec*)
		DTmsec : ARRAY[1..LOGBOOK_ENTRIES_MAX]OF UDINT; (*Additional milliseconds*)
		Severity : ARRAY[1..LOGBOOK_ENTRIES_MAX]OF USINT; (*Severity*)
		Code : ARRAY[1..LOGBOOK_ENTRIES_MAX]OF UINT; (*Code*)
		FacilityCode : ARRAY[1..LOGBOOK_ENTRIES_MAX]OF UINT; (*Facility code*)
		LogbookName : ARRAY[1..LOGBOOK_ENTRIES_MAX]OF STRING[30]; (*Logbook text*)
		ErrorNo : ARRAY[1..LOGBOOK_ENTRIES_MAX]OF DINT; (*Error number*)
		ErrorText : ARRAY[1..LOGBOOK_ENTRIES_MAX]OF STRING[LOGBOOK_TEXT_LEN]; (*Error text*)
	END_STRUCT;
	LogBookCmdType : 	STRUCT  (*Command structure*)
		Refresh : BOOL; (*Read all entries*)
		Update : BOOL; (*Update entries*)
		Create : BOOL; (*Create a new entry*)
		ResetError : BOOL; (*Reset error*)
	END_STRUCT;
	LogBookSegErrorType : 	STRUCT
		ParaSegFilter : STRING[8]; (*show only entries with names beginning with this string*)
		Message : STRING[256]; (*message ArEventLog handling*)
		Record : ARRAY[0..500]OF LogBookSegErrorRecordType;
	END_STRUCT;
	LogBookSegErrorRecordType : 	STRUCT
		ObjectID : STRING[36]; (*logger entry "Entered by"*)
		EventID : DINT; (*logger entry "ID"*)
		EventIDSeverity : USINT; (*logger entry "Severity"*)
		EventIDFacility : UINT; (*logger entry "Facility"*)
		EventIDCode : UINT; (*logger entry "Code"*)
		EventTimeStamp : TIME; (*logger entry "Time"*)
		Text : STRING[300]; (*logger entry "Description"*)
		Description : STRING[256]; (*logger entry "Description"*)
	END_STRUCT;
	LogBookCtrlType : 	STRUCT  (*Main structure*)
		Cmd : LogBookCmdType;
		Par : LogBookParType;
		Data : LogBookDataType;
		Error : LogBookErrorType;
		SegError : LogBookSegErrorType;
		Status : DINT;
		StatusText : STRING[80];
	END_STRUCT;
END_TYPE
```

### TrackDiagGlobal.var
```iecst
VAR CONSTANT
	NUM_HUBS : USINT := 5;
	NUM_PS : USINT := 5;
END_VAR
VAR
	TrackDiag : DiagStatusType;
	paperOptions : TrkPaperCoreOptionsType;
END_VAR
(*LogBook variables*)
VAR
	LogbookInterface : LogBookCtrlType; (*Logbook main structure*)
END_VAR
VAR CONSTANT
	LOGBOOK_EXECUTIONS : USINT := 10; (*Executions per cycle*)
	LOGBOOK_ENTRIES_MAX : UINT := 100; (*Total number of entries*)
	LOGBOOK_BOOKS_MAX : USINT := 13; (*Total number of facilities*)
	LOGBOOK_TEXT_LEN : UINT := 200; (*Error text length*)
END_VAR
(*Module definitions*)
VAR
	DiagInterface : ModuleInterfaceType;
	ModuleName : STRING[40];
END_VAR
```

### Program Logical/Source/SampleTrak/Diagnostic/DiagConfig (IEC)

#### Init.st - Init code
```iecst
PROGRAM _INIT
	(* Insert code here *)

		(* Insert code here *)
	ModuleName := 'DiagModule';

	gRecipeXml_DiagModule;

//	#ifdef ASSEMBLY_STANDARD
//	(*All segment references must be included in the following segment array*)
//	aSegName[0] := gSeg_A_1; 		ErroredSegments[0].SegName := 'gSeg_A_1';
//	aSegName[1] := gSeg_A_2;		ErroredSegments[1].SegName := 'gSeg_A_2';
//	aSegName[2] := gSeg_A_3;		ErroredSegments[2].SegName := 'gSeg_A_3';
//	aSegName[3] := gSeg_A_4;		ErroredSegments[3].SegName := 'gSeg_A_4';
//	aSegName[4] := gSeg_A_5;		ErroredSegments[4].SegName := 'gSeg_A_5';
//	aSegName[5] := gSeg_A_6;		ErroredSegments[5].SegName := 'gSeg_A_6';
//	aSegName[6] := gSeg_A_7;		ErroredSegments[6].SegName := 'gSeg_A_7';
//	aSegName[7] := gSeg_A_8;		ErroredSegments[7].SegName := 'gSeg_A_8';
//	aSegName[8] := gSeg_A_9;		ErroredSegments[8].SegName := 'gSeg_A_9';
//	aSegName[9] := gSeg_A_10;		ErroredSegments[9].SegName := 'gSeg_A_10';
//	aSegName[10] := gSeg_A_11;		ErroredSegments[10].SegName := 'gSeg_A_11';
//	aSegName[11] := gSeg_A_12;		ErroredSegments[11].SegName := 'gSeg_A_12';
//	#endif
//

//	#ifdef ASSEMBLY_STANDARD
//		(*All segment references must be included in the following segment array*)
//		gSegTraceIf.Pars.Segments[0] := ADR(gSeg_A_1 );			segTraceResults[0].SegmentName := 'gSeg_A_1 ';
//		gSegTraceIf.Pars.Segments[1] := ADR(gSeg_A_2 );			segTraceResults[1].SegmentName := 'gSeg_A_2 ';
//		gSegTraceIf.Pars.Segments[2] := ADR(gSeg_A_3 );			segTraceResults[2].SegmentName := 'gSeg_A_3 ';
//		gSegTraceIf.Pars.Segments[3] := ADR(gSeg_A_4 );			segTraceResults[3].SegmentName := 'gSeg_A_4 ';
//		gSegTraceIf.Pars.Segments[4] := ADR(gSeg_A_5 );			segTraceResults[4].SegmentName := 'gSeg_A_5 ';
//		gSegTraceIf.Pars.Segments[5] := ADR(gSeg_A_6 );			segTraceResults[5].SegmentName := 'gSeg_A_6 ';
//		gSegTraceIf.Pars.Segments[6] := ADR(gSeg_A_7 );			segTraceResults[6].SegmentName := 'gSeg_A_7 ';
//		gSegTraceIf.Pars.Segments[7] := ADR(gSeg_A_8 );			segTraceResults[7].SegmentName := 'gSeg_A_8 ';
//		gSegTraceIf.Pars.Segments[8] := ADR(gSeg_A_9 );			segTraceResults[8].SegmentName := 'gSeg_A_9 ';
//		gSegTraceIf.Pars.Segments[9] := ADR(gSeg_A_10);			segTraceResults[9].SegmentName := 'gSeg_A_10';
//		gSegTraceIf.Pars.Segments[10] :=ADR(gSeg_A_11);			segTraceResults[10].SegmentName :='gSeg_A_11';
//		gSegTraceIf.Pars.Segments[11] :=ADR(gSeg_A_12);			segTraceResults[11].SegmentName :='gSeg_A_12';
//
//		gSegTraceIf.Pars.SegmentCount := 12;
//	#endif

END_PROGRAM
```

### Program Logical/Source/SampleTrak/Diagnostic/DiagAlarm (IEC)

#### Variables.var
```iecst
VAR
	fbAlarmDiagModule : MpAlarmXCore;
	FilterConfiguration : STRING[1000] := '';
	SortConfiguration : STRING[1000] := '';
	HistoryFilter : STRING[2000] := '';
	HistorySort : STRING[2000] := '';
	TriggerTestAlarm : BOOL;
	TriggerTestWarning : BOOL;
	TriggerTestInformation : BOOL;
END_VAR
```

### Program Logical/Source/SampleTrak/Diagnostic/TrackDiag (IEC)

#### Main.st - Init, cyclic, exit code
```iecst
PROGRAM _INIT

(* parameter setup for TrackMap *)

	paperCore.SegmentCount := TrackDiag.Seg.SegCount;

	paperCore.Segments := ADR(TrackDiag.Seg.SegList);

	paperCore.Options := ADR(paperOptions);

	paperCore.Enable := TRUE;

(* parameter setup for TrackDiag *)

	AsmReadStatus.Assembly := ADR(DiagInterface.SampleTrak);
	AsmReadInfo.Assembly 	:= ADR(DiagInterface.SampleTrak);

END_PROGRAM

PROGRAM _CYCLIC

	MC_BR_SegCommandError_AcpTrak_0(Segment := ADR(TrackDiag.Seg.SegList[0].McType));

	IF MC_BR_SegCommandError_AcpTrak_0.Done THEN
		MC_BR_SegCommandError_AcpTrak_0.Execute := FALSE;
	END_IF

	(***********************************ASSEMBLY INFORMATION******************************	)
	(*Read Assebly Status*)

	AsmReadStatus.Enable	:= TRUE;
	AsmReadStatus();

	IF AsmReadStatus.Valid THEN
		TrackDiag.Asm.AssemblyDisabled 	:= AsmReadStatus.AssemblyDisabled;
		TrackDiag.Asm.AssemblyErrorStop := AsmReadStatus.AssemblyErrorStop;
		TrackDiag.Asm.AssemblyReady		:= AsmReadStatus.AssemblyReady;
		TrackDiag.Asm.AssemblyHoming	:= AsmReadStatus.AssemblyHoming;
		TrackDiag.Asm.AssemblyStopping	:= AsmReadStatus.AssemblyStopping;
	END_IF

	(*Read Assembly Info *)

	AsmReadInfo.Enable		:= TRUE;
	AsmReadInfo();

	IF AsmReadInfo.Valid THEN
		TrackDiag.Asm.CommunicationReady 	:= AsmReadInfo.AssemblyInfo.CommunicationReady;
		TrackDiag.Asm.PowerOn				:= AsmReadInfo.AssemblyInfo.PowerOn;
		TrackDiag.Asm.ReadyForPowerOn		:= AsmReadInfo.AssemblyInfo.ReadyForPowerOn;
		TrackDiag.Asm.ShuttleInErrorStopCount := AsmReadInfo.AssemblyInfo.ShuttlesInErrorStopCount;
		TrackDiag.Asm.StartupCount			:= AsmReadInfo.AssemblyInfo.StartupCount;
	END_IF

	(****************************** SEGMENT ERROR INFORMATION *****************************************)

	FOR SegIndex := 0 TO NUM_SEG DO

		IF TrackDiag.Seg.SegList[SegIndex].McType.controlif <> 0 THEN //If the array contains a segment reference
			SegReadInfo[SegIndex].Segment 	:= ADR(TrackDiag.Seg.SegList[SegIndex].McType);
			SegReadInfo[SegIndex].Enable	:= TRUE;
			SegReadInfo[SegIndex]();

			IF SegReadInfo[SegIndex].Valid THEN
				//Capture Segment Info
				TrackDiag.Seg.SegList[SegIndex].Status.CommunicationReady 	:= SegReadInfo[SegIndex].SegmentInfo.CommunicationReady;
				TrackDiag.Seg.SegList[SegIndex].Status.ReadyForPowerOn		:= SegReadInfo[SegIndex].SegmentInfo.ReadyForPowerOn;
				TrackDiag.Seg.SegList[SegIndex].Status.PowerOn				:= SegReadInfo[SegIndex].SegmentInfo.PowerOn;
				TrackDiag.Seg.SegList[SegIndex].Status.StartupCount			:= SegReadInfo[SegIndex].SegmentInfo.StartupCount;
				TrackDiag.Seg.SegList[SegIndex].Status.CommunicationState	:= SegReadInfo[SegIndex].SegmentInfo.CommunicationState;

			END_IF

			SegReadStatus[SegIndex].Segment := ADR(TrackDiag.Seg.SegList[SegIndex].McType);
			SegReadStatus[SegIndex].Enable	:= TRUE;
			SegReadStatus[SegIndex]();

			IF SegReadStatus[SegIndex].Valid THEN

				//Check for change of state to ErrorStop to command reading error data, IF communication is ready
				IF ((TrackDiag.Seg.SegList[SegIndex].Status.SegmentErrorStop = FALSE AND SegReadStatus[SegIndex].SegmentErrorStop = TRUE))
					AND (TrackDiag.Seg.SegList[SegIndex].Status.CommunicationReady = TRUE) THEN

					SegErrorCheck[SegIndex].CmdCheckErrorCode := TRUE;

					//Check for change of state from ErrorStop to reset error number in diag structure
				ELSIF ((TrackDiag.Seg.SegList[SegIndex].Status.SegmentErrorStop = TRUE) AND (SegReadStatus[SegIndex].SegmentErrorStop = FALSE))
					AND (TrackDiag.Seg.SegList[SegIndex].Status.CommunicationReady = TRUE) THEN

					TrackDiag.Seg.SegList[SegIndex].Status.ErrorCode := 0;

				END_IF
				//Capture Segment Status

				TrackDiag.Seg.SegList[SegIndex].Status.SegmentDisabled	:= SegReadStatus[SegIndex].SegmentDisabled;
				TrackDiag.Seg.SegList[SegIndex].Status.SegmentErrorStop	:= SegReadStatus[SegIndex].SegmentErrorStop;
				TrackDiag.Seg.SegList[SegIndex].Status.SegmentReady		:= SegReadStatus[SegIndex].SegmentReady;
				TrackDiag.Seg.SegList[SegIndex].Status.SegmentStopping	:= SegReadStatus[SegIndex].SegmentStopping;
			END_IF
		END_IF
	END_FOR

	CpuSim := DiagCpuIsSimulated() OR DiagCpuIsARsim();

	IF CpuSim = FALSE THEN
		actCheckErrorCode;
	END_IF

	fbAuditTrail(MpLink := ADR(gAuditTrail_DiagModule), Enable := TRUE, Language := ADR('en'), DeviceName := ADR('User'));

	(***********************************TRACKMAP******************************)

	paperCore();

	// compare the elementID clicked on in paper with the configured ID to find and set the array index for the list binding
	FOR SegIndex:= 0 TO NUM_SEG DO

		// clickId contains a leading # which needs to be removed,
		// the second compare checks against the text and arrow and deletes the first two letters because the SVG elements text and arrow have an added x leading the name
		IF TrackDiag.Seg.SegList[SegIndex].Name = DELETE(clickId,1,1) OR TrackDiag.Seg.SegList[SegIndex].Name = DELETE(clickId,1,2)THEN
			clickedSegment := TrackDiag.Seg.SegList[SegIndex];
			EXIT;
		END_IF
	END_FOR
END_PROGRAM

PROGRAM _EXIT
			(* Insert code here *)

END_PROGRAM
```

#### Types.typ - Local data types
```iecst
TYPE
	CheckStateEnum :
		(
		WAIT_FOR_CHECK,
		READ_DATA,
		READ_DATA_SEG_STATE,
		CHECK_SEG_STATE,
		READ_DATA_SEG_ERROR_STAT,
		CHECK_ERROR_STAT,
		READ_DATA_SEG_ERROR,
		CHECK_ERROR_CODE,
		WRITE_WARNING_CODE,
		READ_DATA_SEG_LAG,
		CHECK_SEG_LAG,
		READ_DATA_SEG_VEL,
		CHECK_SEG_VEL,
		READ_DATA_SEG_TEMP,
		CHECK_DATA_SEG_TEMP,
		WRITE_SPEED_FILTER,
		WRITE_SPEED_FILTER_WAIT,
		WRITE_ZERO_PITCH,
		READ_EXEC_ERROR,
		READ_SEG_STATUS,
		WRITE_SEG_RESET,
		WAIT_FOR_DONE
		);
	SegErrorCheckType : 	STRUCT
		CheckState : CheckStateEnum;
		CmdCheckErrorCode : BOOL;
		DataReadExecutionError : BOOL;
		ErrorNumber : UINT;
		SegStatusBits : UDINT;
		ErrorStatusBit : BOOL;
		ErrorStatus : UDINT;
	END_STRUCT;
	SegShuttleMonitorType : 	STRUCT
		CheckState_enum : BOOL;
		CmdMonitorLag : BOOL;
		CmdMonitorVelocity : BOOL;
		Lag : ARRAY[0..2]OF LREAL;
		Velocity : ARRAY[0..2]OF LREAL;
		LagLimitExceeded : BOOL;
		VelLimitExceeded : BOOL;
	END_STRUCT;
	SegTempCheckType : 	STRUCT
		CheckState : CheckStateEnum;
		CmdCheckTemp : BOOL;
		DataReadExecutionError : BOOL;
	END_STRUCT;
	SegPitchSetType : 	STRUCT
		CheckState : CheckStateEnum;
		CmdSetPitch : BOOL;
		CmdWriteFilter : BOOL;
		PitchSetComplete : BOOL;
		FilterWriteComplete : BOOL;
		DataReadExecutionError : BOOL;
		ErrorID : UDINT;
	END_STRUCT;
END_TYPE
```

#### Variables.var - Local variables
```iecst
VAR
	AsmReadInfo : MC_BR_AsmReadInfo_AcpTrak;
	AsmReadStatus : MC_BR_AsmReadStatus_AcpTrak;
	SegReadInfo : ARRAY[0..NUM_SEG] OF MC_BR_SegReadInfo_AcpTrak;
	SegReadStatus : ARRAY[0..NUM_SEG] OF MC_BR_SegReadStatus_AcpTrak;
	SegIndex : USINT;
	SegProcessParID : ARRAY[0..NUM_SEG] OF MC_BR_SegProcessParID_AcpTrak;
	ErrorCodeIDInfo : ARRAY[0..NUM_SEG] OF McAcpTrakSegProcessParIDType;
	SegWarningCmdIDInfo : McAcpTrakSegProcessParIDType;
	SegErrorCheck : ARRAY[0..NUM_SEG] OF SegErrorCheckType;
	CmdWarning : UINT;
	Current : ARRAY[0..20] OF INT; (*Power Supply Current*)
	Voltage : ARRAY[0..20] OF SINT; (*Power Supply Voltage*)
	fbAuditTrail : MpAuditTrail;
	CpuSim : BOOL;
END_VAR
(*For testing only*)
VAR
	MC_BR_SegCommandError_AcpTrak_0 : MC_BR_SegCommandError_AcpTrak;
END_VAR
(*Declarations for TrackMap*)
VAR
	paperCore : TrkPaperCore;
	clickId : STRING[160];
	clickedSegment : TrkDiagSegmentType;
END_VAR
```

#### CheckErrorCode.st
```iecst
ACTION actCheckErrorCode:

	FOR SegIndex := 0 TO NUM_SEG DO

		CASE SegErrorCheck[SegIndex].CheckState OF

			WAIT_FOR_CHECK:
				//Wait for the command to check the error code ParID on the segment
				SegProcessParID[SegIndex].Execute := FALSE;

				IF SegErrorCheck[SegIndex].CmdCheckErrorCode THEN
					SegProcessParID[SegIndex].Execute := TRUE;
//					SegProcessParID[SegIndex].DataAddress := ADR(SegStateIDInfo[SegIndex]);
//					SegErrorCheck[SegIndex].CheckState := READ_DATA_SEG_STATE;
					SegProcessParID[SegIndex].Mode := mcACPTRAK_SEG_PARID_GET_NO_NCT;
					SegProcessParID[SegIndex].DataAddress := ADR(ErrorCodeIDInfo[SegIndex]);
					SegErrorCheck[SegIndex].CheckState := READ_DATA_SEG_ERROR;
					SegErrorCheck[SegIndex].CmdCheckErrorCode := FALSE; //Reset check command

				END_IF

			READ_DATA_SEG_ERROR:
				//Check for completion of reading the PARID for

				IF SegProcessParID[SegIndex].Done THEN
					//If the parID was successfully read, go to check error code state
					SegErrorCheck[SegIndex].CheckState := CHECK_ERROR_CODE;
					SegProcessParID[SegIndex].Execute := FALSE;
					SegErrorCheck[SegIndex].DataReadExecutionError := FALSE;

				ELSIF SegProcessParID[SegIndex].Error THEN
					//If there was an error in reading, go to error start
					SegErrorCheck[SegIndex].CheckState := READ_EXEC_ERROR;
				END_IF

			CHECK_ERROR_CODE:

				IF (SegErrorCheck[SegIndex].ErrorNumber = 0) OR (SegErrorCheck[SegIndex].ErrorNumber = 36005) THEN
					//Segment has no new error recorded. Shows either 0 or the commanded warning (36005) used to overwrite old errors
					TrackDiag.Seg.SegList[SegIndex].Status.ErrorCode := 0;
					SegErrorCheck[SegIndex].CheckState := WAIT_FOR_CHECK;
					TrackDiag.Seg.SegList[SegIndex].Status.Error := FALSE;

				ELSE
					//Otherwise, there is a new error on this segment
					TrackDiag.Seg.SegList[SegIndex].Status.ErrorCode := SegErrorCheck[SegIndex].ErrorNumber;

					TrackDiag.Seg.SegList[SegIndex].Status.Error := TRUE;
					//Send to overwrite state to store a known error number (36005) in the error code parID
					SegErrorCheck[SegIndex].CheckState := WRITE_WARNING_CODE;

					//Send data to HMI
					IF(SegIndex > 0)THEN

						ErrorSegNum[ErrorCnt] 	:= SegIndex - 1;
						ErrorSegName[ErrorCnt]	:= TrackDiag.Seg.SegList[SegIndex].Name;
						ErrorNumber[ErrorCnt]	:= TrackDiag.Seg.SegList[SegIndex].Status.ErrorCode;
						ErrorCnt := ErrorCnt + 1;

					END_IF

				END_IF

			WRITE_WARNING_CODE:
				//Write commanded warning code (36005) to error parid
				SegProcessParID[SegIndex].DataAddress := ADR(SegWarningCmdIDInfo);
				SegProcessParID[SegIndex].ChannelIndex := 0;
				SegProcessParID[SegIndex].Mode := mcACPTRAK_SEG_PARID_SET;
				SegProcessParID[SegIndex].NumberOfParIDs := 0;
				SegProcessParID[SegIndex].Execute := TRUE;

				IF SegProcessParID[SegIndex].Done THEN
					//return to wait state
					SegProcessParID[SegIndex].Execute := FALSE;
					SegErrorCheck[SegIndex].CheckState := WAIT_FOR_CHECK;

				ELSIF SegProcessParID[SegIndex].Error THEN
					SegErrorCheck[SegIndex].CheckState := READ_EXEC_ERROR;
				END_IF

			READ_EXEC_ERROR:
				SegProcessParID[SegIndex].Execute := FALSE;
				SegErrorCheck[SegIndex].DataReadExecutionError := TRUE;

				IF SegProcessParID[SegIndex].Error = FALSE THEN
					SegErrorCheck[SegIndex].CheckState := WAIT_FOR_CHECK;
				END_IF

		END_CASE

	SegProcessParID[SegIndex]();
	END_FOR

END_ACTION
```

#### CheckTemp.st
```iecst
ACTION actCheckTemp:

	FOR SegIndex := 0 TO NUM_SEG DO

		CASE SegTempCheck[SegIndex].CheckState OF

			WAIT_FOR_CHECK:
				//Wait for the command to check the the temperature data on the motor segment
				SegProcessParID_Temp[SegIndex].Execute := FALSE;

				IF SegTempCheck[SegIndex].CmdCheckTemp THEN
					SegTempCheck[SegIndex].CheckState := READ_DATA_SEG_TEMP;
					SegProcessParID_Temp[SegIndex].Execute := TRUE;
					SegTempCheck[SegIndex].CmdCheckTemp := FALSE; //Reset check command
				END_IF

			READ_DATA_SEG_TEMP:
				//Check for completion of reading Segment Status Bits
				IF SegProcessParID_Temp[SegIndex].Done THEN

					//If the parID was successfully read, go to check seg state
					SegTempCheck[SegIndex].CheckState := WAIT_FOR_CHECK;
					SegProcessParID_Temp[SegIndex].Execute := FALSE;
					SegTempCheck[SegIndex].DataReadExecutionError := FALSE;

				ELSIF SegProcessParID_Temp[SegIndex].Error THEN
					//If there was an error in reading, go to error start
					SegTempCheck[SegIndex].CheckState := READ_EXEC_ERROR;
				END_IF

			CHECK_DATA_SEG_TEMP:

			READ_EXEC_ERROR:
				SegProcessParID_Temp[SegIndex].Execute := FALSE;
				SegTempCheck[SegIndex].DataReadExecutionError := TRUE;

				IF SegProcessParID_Temp[SegIndex].Error = FALSE THEN
					SegTempCheck[SegIndex].CheckState := WAIT_FOR_CHECK;
				END_IF

		END_CASE

		SegProcessParID_Temp[SegIndex]();
	END_FOR

END_ACTION
```

#### TrakLogger.typ - not listed in the package file held
```iecst
(*read & filter motion logger*)

TYPE
	TrakLoggerType : 	STRUCT
		CmdRefresh : BOOL; (*command read & filter motion logger*)
		ParaShowSegError : BOOL; (*filter - show motion logger enties severity error*)
		ParaShowSegWarning : BOOL; (*filter - show motion logger enties severity warning*)
		ParaSegFilter : STRING[8]; (*show only entries with names beginning with this string*)
		Message : STRING[256]; (*message ArEventLog handling*)
		Record : ARRAY[0..500]OF TrakLoggerRecordType;
	END_STRUCT;
	TrakLoggerRecordType : 	STRUCT
		ObjectID : STRING[36]; (*logger entry "Entered by"*)
		EventID : DINT; (*logger entry "ID"*)
		EventIDSeverity : USINT; (*logger entry "Severity"*)
		EventIDFacility : UINT; (*logger entry "Facility"*)
		EventIDCode : UINT; (*logger entry "Code"*)
		EventTimeStamp : TIME; (*logger entry "Time"*)
		Text : STRING[300]; (*logger entry "Description"*)
		Description : STRING[256]; (*logger entry "Description"*)
	END_STRUCT;
END_TYPE

(*enum*)

TYPE
	StepEnum :
		(
		TRAK_COMMAND := 0,
		TRAK_RESET,
		TRAK_GET_IDENT := 10,
		TRAK_GET_IDENT_WAIT,
		TRAK_GET_LATEST_ID,
		TRAK_GET_LATEST_ID_WAIT,
		TRAK_GET_PREVIOUS_ID := 20,
		TRAK_GET_PREVIOUS_ID_WAIT,
		TRAK_READ_ID := 30,
		TRAK_READ_ID_WAIT,
		TRAK_CHECK_FILTER := 40,
		TRAK_CHECK_FILTER_WAIT,
		TRAK_READ_DESCRIPTION := 50,
		TRAK_READ_DESCRIPTION_WAIT,
		TRAK_UPDATE_LIST := 60,
		TRAK_DONE := 90,
		TRAK_ERROR := 99
		);
END_TYPE
```

#### TrakLogger.var - not listed in the package file held
```iecst
(*read & filter motion logger*)
VAR
	TrakLogger : TrakLoggerType;
	Step : StepEnum := (0);
	StepLast : StepEnum := (0);
	Ident : ArEventLogIdentType := (0);
	RecordID : ArEventLogRecordIDType := (0);
	EventTimeStamp : ArEventLogTimeStampType := (0);
	EventID : DINT := 0;
	EventIDSeverity : USINT := 0;
	EventIDFacility : UINT := 0;
	EventIDCode : UINT := 0;
	ObjectID : STRING[36] := '';
	Description : STRING[256] := '';
	TempString : STRING[32] := '';
	SegmentErrorFound : USINT := 0;
	AlarmCount : ARRAY[0..119] OF UDINT;
	TimeStruct : TIMEStructure;
	FirstEntryCheckSum : USINT;
END_VAR
(*ArEventLog FUB*)
VAR
	FubTonWaitFirst : TON := (0);
	ArEventLogGetIdent_0 : ArEventLogGetIdent := (0);
	ArEventLogGetLatestRecordID_0 : ArEventLogGetLatestRecordID := (0);
	ArEventLogGetPreviousRecordID_0 : ArEventLogGetPreviousRecordID := (0);
	ArEventLogRead_0 : ArEventLogRead := (0);
	ArEventLogReadObjectID_0 : ArEventLogReadObjectID := (0);
	ArEventLogReadDescription_0 : ArEventLogReadDescription := (0);
END_VAR
(*Test function*)
VAR
	MC_BR_SegCommandError_AcpTrak_0 : MC_BR_SegCommandError_AcpTrak;
END_VAR
```

#### SegmentReset.st - not listed in the package file held
```iecst
ACTION actSegmentReset:

	FOR SegIndex := 0 TO NUM_SEG DO

		CASE SegmentReset[SegIndex].State OF

			WAIT_FOR_CHECK:

				//Wait for the command to check the segment status
				SegProcessParID_Reset[SegIndex].Execute := FALSE;

				IF SegmentReset[SegIndex].CmdResetSeg THEN

					SegmentReset[SegIndex].CmdResetSeg 		:= FALSE; //Reset check command
					SegmentReset[SegIndex].StsResetDone 	:= FALSE; //Reset done status

					//Check segment status
					IF NOT(SegReadInfo[SegIndex].SegmentInfo.ReadyForPowerOn)THEN

						IF(TrackDiag.Seg.SegList[SegIndex].Status.ErrorCode = 6020)THEN  		//Undervoltage error
							SegmentReset[SegIndex].State := WRITE_SEG_RESET;
						ELSE
							SegmentReset[SegIndex].State := WAIT_FOR_DONE;
						END_IF

					ELSE

						SegmentReset[SegIndex].State 	:= WAIT_FOR_DONE;

					END_IF

				END_IF

			WRITE_SEG_RESET:

				//Wait for the command to check the error code ParID on the segment
				SegProcessParID_Reset[SegIndex].Execute := TRUE;
				SegProcessParID_Reset[SegIndex].Mode 	:= mcACPTRAK_SEG_PARID_SET;
				SegProcessParID_Reset[SegIndex].DataAddress := ADR(SegResetIDInfo[SegIndex]);

				//Check for completion of reading the PARID for
				IF SegProcessParID_Reset[SegIndex].Done THEN
					//If the parID was successfully read, go to check error code state
					SegProcessParID_Reset[SegIndex].Execute 		:= FALSE;
					SegmentReset[SegIndex].DataReadExecutionError 	:= FALSE;

					SegmentReset[SegIndex].State 			:= WAIT_FOR_DONE;

				ELSIF SegProcessParID_Reset[SegIndex].Error THEN
					//If there was an error in reading, go to error start
					SegmentReset[SegIndex].State := READ_EXEC_ERROR;
				END_IF

			WAIT_FOR_DONE:

				IF (SegReadInfo[SegIndex].SegmentInfo.ReadyForPowerOn)THEN

					SegmentReset[SegIndex].StsResetDone 	:= TRUE; //Set done status
					SegmentReset[SegIndex].State 			:= WAIT_FOR_CHECK;

				ELSIF SegReadInfo[SegIndex].Error THEN
					//If there was an error in reading, go to error start
					SegmentReset[SegIndex].State := READ_EXEC_ERROR;

				END_IF

			READ_EXEC_ERROR:
				SegProcessParID_Reset[SegIndex].Execute := FALSE;
				SegmentReset[SegIndex].DataReadExecutionError := TRUE;

				IF SegProcessParID_Reset[SegIndex].Error = FALSE THEN
					SegmentReset[SegIndex].State := WAIT_FOR_CHECK;
				END_IF

		END_CASE

		SegProcessParID_Reset[SegIndex]();
	END_FOR

END_ACTION
```

#### TrakLogger.st - not listed in the package file held
```iecst
ACTION TrakLoggerInit:

	TrakLogger.CmdRefresh			:= FALSE;
	TrakLogger.ParaShowSegError		:= TRUE;
	TrakLogger.ParaShowSegWarning	:= TRUE;
	TrakLogger.ParaSegFilter		:= 'Asm';//'gSeg_';

	Step := TRAK_COMMAND;

END_ACTION

ACTION TrakLoggerCyclic:

	MC_BR_SegCommandError_AcpTrak_0(Segment := ADR(TrackDiag.Seg.SegList[0].McType));

	IF MC_BR_SegCommandError_AcpTrak_0.Done THEN
		MC_BR_SegCommandError_AcpTrak_0.Execute := FALSE;
	END_IF

	IF EDGEPOS(TrackDiag.Asm.AssemblyErrorStop) THEN
		TrakLogger.CmdRefresh := TRUE;
	END_IF

	REPEAT
		StepLast := Step;

		CASE Step OF

			//////////////////////////////////////////////////////////////////////////////////////////////////////////////////////////////
			// command
			TRAK_COMMAND:
				IF TrakLogger.CmdRefresh THEN
					Step := TRAK_RESET;
				END_IF

			//////////////////////////////////////////////////////////////////////////////////////////////////////////////////////////////
			// wait till all messages are entered into logger
			TRAK_RESET:
				FubTonWaitFirst.IN := TRUE;
				FubTonWaitFirst.PT := T#1s;
				FubTonWaitFirst();
				IF FubTonWaitFirst.Q THEN
					FubTonWaitFirst.IN := FALSE;

					brsmemset(ADR(TrakLogger.Record), 0, SIZEOF(TrakLogger.Record));
					TrakLogger.Message := '';
					SegmentErrorFound := 0;

					brsmemset(ADR(AlarmCount), 0, SIZEOF(AlarmCount));

					ArEventLogGetIdent_0.Execute			:= FALSE;
					ArEventLogGetLatestRecordID_0.Execute	:= FALSE;
					ArEventLogGetPreviousRecordID_0.Execute	:= FALSE;
					ArEventLogRead_0.Execute				:= FALSE;
					ArEventLogReadObjectID_0.Execute		:= FALSE;
					ArEventLogReadDescription_0.Execute		:= FALSE;
					Step := TRAK_GET_IDENT;
				END_IF

			///////////////////////////////////////////////////////////////////////////
			// open logger and read first EventID
			TRAK_GET_IDENT:
				ArEventLogGetIdent_0.Execute	:= TRUE;
				brsstrcpy(ADR(ArEventLogGetIdent_0.Name), ADR('$$motion'));
				Step := TRAK_GET_IDENT_WAIT;

			TRAK_GET_IDENT_WAIT:
				IF ArEventLogGetIdent_0.Done THEN
					Ident := ArEventLogGetIdent_0.Ident;
					ArEventLogGetIdent_0.Execute := FALSE;
					Step := TRAK_GET_LATEST_ID;
				ELSIF ArEventLogGetIdent_0.Error THEN
					TrakLogger.Message := 'Error GetIdent';
					Step := TRAK_ERROR;
				END_IF

			TRAK_GET_LATEST_ID:
				ArEventLogGetLatestRecordID_0.Execute	:= TRUE;
				ArEventLogGetLatestRecordID_0.Ident		:= Ident;
				Step := TRAK_GET_LATEST_ID_WAIT;

			TRAK_GET_LATEST_ID_WAIT:
				IF ArEventLogGetLatestRecordID_0.Done THEN
					RecordID := ArEventLogGetLatestRecordID_0.RecordID;
					ArEventLogGetLatestRecordID_0.Execute := FALSE;
					Step := TRAK_READ_ID;
				ELSIF ArEventLogGetLatestRecordID_0.Error THEN
					TrakLogger.Message := 'Error GetLatestRecordID';
					Step := TRAK_ERROR;
				END_IF

			///////////////////////////////////////////////////////////////////////////
			// read previous EventID
			TRAK_GET_PREVIOUS_ID:
				ArEventLogGetPreviousRecordID_0.Execute		:= TRUE;
				ArEventLogGetPreviousRecordID_0.Ident		:= Ident;
				ArEventLogGetPreviousRecordID_0.RecordID	:= RecordID;
				Step := TRAK_GET_PREVIOUS_ID_WAIT;

			TRAK_GET_PREVIOUS_ID_WAIT:
				IF ArEventLogGetPreviousRecordID_0.Done THEN
					RecordID := ArEventLogGetPreviousRecordID_0.PrevRecordID;
					ArEventLogGetPreviousRecordID_0.Execute := FALSE;
					Step := TRAK_READ_ID;
				ELSIF ArEventLogGetPreviousRecordID_0.Error THEN
					IF ArEventLogGetPreviousRecordID_0.StatusID = arEVENTLOG_ERR_RECORDID_INVALID THEN		// reached end of logger
						ArEventLogGetPreviousRecordID_0.Execute := FALSE;
						Step := TRAK_DONE;
					ELSE
						TrakLogger.Message := 'Error GetPreviousRecordID';
						Step := TRAK_ERROR;
					END_IF
				END_IF

			///////////////////////////////////////////////////////////////////////////
			// check if severity is 'Error' or 'Warning'
			TRAK_READ_ID:
				ArEventLogRead_0.Execute	:= TRUE;
				ArEventLogRead_0.Ident		:= Ident;
				ArEventLogRead_0.RecordID	:= RecordID;
				Step := TRAK_READ_ID_WAIT;

			TRAK_READ_ID_WAIT:
				IF ArEventLogRead_0.Done THEN
					EventID := ArEventLogRead_0.EventID;
					ArEventLogRead_0.Execute := FALSE;
					EventTimeStamp := ArEventLogRead_0.TimeStamp;

					EventIDSeverity	:= DINT_TO_USINT(SHR(EventID, 30) AND 16#03);
					EventIDFacility	:= DINT_TO_UINT(SHR(EventID, 16) AND 16#0FFF);
					EventIDCode		:= DINT_TO_UINT(SHR(EventID, 0) AND 16#FFFF);

					IF ((EventIDSeverity = arEVENTLOG_SEVERITY_ERROR) AND (TrakLogger.ParaShowSegError)) THEN
						Step := TRAK_CHECK_FILTER;
					ELSIF ((EventIDSeverity = arEVENTLOG_SEVERITY_WARNING) AND (TrakLogger.ParaShowSegWarning)) THEN
						Step := TRAK_CHECK_FILTER;
					ELSE
						Step := TRAK_GET_PREVIOUS_ID;
					END_IF
				ELSIF ArEventLogRead_0.Error THEN
					TrakLogger.Message := 'Error ReadRecordID';
					Step := TRAK_ERROR;
				END_IF

			///////////////////////////////////////////////////////////////////////////
			// check if 'Error' has been entered by a Segment
			TRAK_CHECK_FILTER:
				ArEventLogReadObjectID_0.Execute	:= TRUE;
				ArEventLogReadObjectID_0.Ident		:= Ident;
				ArEventLogReadObjectID_0.RecordID	:= RecordID;
				Step := TRAK_CHECK_FILTER_WAIT;

			TRAK_CHECK_FILTER_WAIT:
				IF ArEventLogReadObjectID_0.Done THEN
					ObjectID := ArEventLogReadObjectID_0.ObjectID;
					ArEventLogReadObjectID_0.Execute := FALSE;
					IF brsmemcmp(ADR(ObjectID), ADR(TrakLogger.ParaSegFilter), 3) = 0 THEN
						Step := TRAK_READ_DESCRIPTION;
					ELSE
						Step := TRAK_GET_PREVIOUS_ID;
					END_IF
				ELSIF ArEventLogReadObjectID_0.Error THEN
					TrakLogger.Message := 'Error ReadObjectID';
					Step := TRAK_ERROR;
				END_IF

			///////////////////////////////////////////////////////////////////////////
			// read and display description text if filter criterias are matching
			TRAK_READ_DESCRIPTION:
				ArEventLogReadDescription_0.Execute			:= TRUE;
				ArEventLogReadDescription_0.Ident			:= Ident;
				ArEventLogReadDescription_0.RecordID		:= RecordID;
			//	ArEventLogReadDescription_0.LanguageCode	:= ;
			//	ArEventLogReadDescription_0.Qualifier		:= ;
				ArEventLogReadDescription_0.TextBuffer		:= ADR(Description);
				ArEventLogReadDescription_0.TextBufferSize	:= SIZEOF(Description);
				Step := TRAK_READ_DESCRIPTION_WAIT;

			TRAK_READ_DESCRIPTION_WAIT:
				IF ArEventLogReadDescription_0.Done THEN
					ArEventLogReadDescription_0.Execute := FALSE;
					Step := TRAK_UPDATE_LIST;
				ELSIF ArEventLogReadDescription_0.Error THEN
					TrakLogger.Message := 'Error ReadDescription';
					Step := TRAK_ERROR;
				END_IF

			TRAK_UPDATE_LIST:
				TrakLogger.Record[SegmentErrorFound].ObjectID			:= ObjectID;
				TrakLogger.Record[SegmentErrorFound].EventID			:= EventID;
				TrakLogger.Record[SegmentErrorFound].EventIDSeverity	:= EventIDSeverity;
				TrakLogger.Record[SegmentErrorFound].EventIDFacility	:= EventIDFacility;
				TrakLogger.Record[SegmentErrorFound].EventIDCode		:= EventIDCode;
				TrakLogger.Record[SegmentErrorFound].Description		:= Description;

				TrakLogger.Record[SegmentErrorFound].EventTimeStamp	:= UDINT_TO_TIME((EventTimeStamp.sec MOD (24*60*60))*1000 + (EventTimeStamp.nsec / 1000000));		// convert to TIME format (ms since start of day)

				brsstrcpy(ADR(TrakLogger.Record[SegmentErrorFound].Text), ADR(''));
				ascTIME(TrakLogger.Record[SegmentErrorFound].EventTimeStamp, ADR(TempString), SIZEOF(TempString));
				TIME_TO_TIMEStructure(TrakLogger.Record[SegmentErrorFound].EventTimeStamp,ADR(TimeStruct)); // for checking against older entries

				brsstrcat(ADR(TrakLogger.Record[SegmentErrorFound].Text), ADR(TempString));
				brsstrcat(ADR(TrakLogger.Record[SegmentErrorFound].Text), ADR(' => '));

				brsstrcat(ADR(TrakLogger.Record[SegmentErrorFound].Text), ADR(ObjectID));

				brsstrcat(ADR(TrakLogger.Record[SegmentErrorFound].Text), ADR(': Error '));
				brsitoa(EventIDCode, ADR(TempString));
				brsstrcat(ADR(TrakLogger.Record[SegmentErrorFound].Text), ADR(TempString));

				brsstrcat(ADR(TrakLogger.Record[SegmentErrorFound].Text), ADR(' => '));
				brsstrcat(ADR(TrakLogger.Record[SegmentErrorFound].Text), ADR(Description));

				IF SegmentErrorFound = 0 THEN
					FirstEntryCheckSum := TimeStruct.minute; // save the timestamp minute of the first entry as checksum
				END_IF

				SegmentErrorFound := SegmentErrorFound + 1;

				SetAlarmIDCode; //case statement to trigger alarms

				// stop reading the logger when the end of the array is reached OR
				// when the entries start having a different timestamp which means they are older
				IF SegmentErrorFound > 499 OR (FirstEntryCheckSum <> (TimeStruct.minute) ) THEN
					Step := TRAK_DONE;
				ELSE
					Step := TRAK_GET_PREVIOUS_ID;
				END_IF

			//////////////////////////////////////////////////////////////////////////////////////////////////////////////////////////////
			TRAK_DONE:
				TrakLogger.CmdRefresh := FALSE;
				Step := TRAK_COMMAND;

			//////////////////////////////////////////////////////////////////////////////////////////////////////////////////////////////
			TRAK_ERROR:
				IF TrakLogger.CmdRefresh = 0 THEN
					TrakLogger.Message := '';
					ArEventLogGetIdent_0.Execute			:= FALSE;
					ArEventLogGetLatestRecordID_0.Execute	:= FALSE;
					ArEventLogGetPreviousRecordID_0.Execute	:= FALSE;
					ArEventLogRead_0.Execute				:= FALSE;
					ArEventLogReadObjectID_0.Execute		:= FALSE;
					ArEventLogReadDescription_0.Execute		:= FALSE;
					Step := TRAK_COMMAND;
				END_IF

		END_CASE

		ArEventLogGetIdent_0();
		ArEventLogGetLatestRecordID_0();
		ArEventLogGetPreviousRecordID_0();
		ArEventLogRead_0();
		ArEventLogReadObjectID_0();
		ArEventLogReadDescription_0();

	UNTIL
		// to speed processing time of this sequence up: repeat sequence till the step is not changing any more (sequence is waiting for a FUB)
		Step = StepLast

	END_REPEAT

END_ACTION

ACTION SetAlarmIDCode:

		// EventIDCode add new alarms triggers at the end otherwise
		// the AlarmCount has to be adjusted not just here but also for all the alarms in the MpAlarmX config

		CASE EventIDCode OF
		// every time the alarm is triggered it's counted so a total count can be displayed in the alarm message
		1	 :  AlarmCount[0  ] :=  AlarmCount[0]  + 1;   MpAlarmXSet(DiagInterface.AlarmCore,'EventIDCode.1	');
		2	 :  AlarmCount[1  ] :=  AlarmCount[1]  + 1;   MpAlarmXSet(DiagInterface.AlarmCore,'EventIDCode.2	');
		7	 :  AlarmCount[2  ] :=  AlarmCount[2]  + 1;   MpAlarmXSet(DiagInterface.AlarmCore,'EventIDCode.7	');
		2048 :  AlarmCount[3  ] :=  AlarmCount[3]  + 1;   MpAlarmXSet(DiagInterface.AlarmCore,'EventIDCode.2048');
		2049 :  AlarmCount[4  ] :=  AlarmCount[4]  + 1;   MpAlarmXSet(DiagInterface.AlarmCore,'EventIDCode.2049');
		2050 :  AlarmCount[5  ] :=  AlarmCount[5]  + 1;   MpAlarmXSet(DiagInterface.AlarmCore,'EventIDCode.2050');
		2051 :  AlarmCount[6  ] :=  AlarmCount[6]  + 1;   MpAlarmXSet(DiagInterface.AlarmCore,'EventIDCode.2051');
		2052 :  AlarmCount[7  ] :=  AlarmCount[7]  + 1;   MpAlarmXSet(DiagInterface.AlarmCore,'EventIDCode.2052');
		2053 :  AlarmCount[8  ] :=  AlarmCount[8]  + 1;   MpAlarmXSet(DiagInterface.AlarmCore,'EventIDCode.2053');
		2054 :  AlarmCount[9  ] :=  AlarmCount[9]  + 1;   MpAlarmXSet(DiagInterface.AlarmCore,'EventIDCode.2054');
		2055 :  AlarmCount[10 ] := AlarmCount[10]  + 1;   MpAlarmXSet(DiagInterface.AlarmCore,'EventIDCode.2055');
		2056 :  AlarmCount[11 ] := AlarmCount[11]  + 1;   MpAlarmXSet(DiagInterface.AlarmCore,'EventIDCode.2056');
		2057 :  AlarmCount[12 ] := AlarmCount[12]  + 1;   MpAlarmXSet(DiagInterface.AlarmCore,'EventIDCode.2057');
		2058 :  AlarmCount[13 ] := AlarmCount[13]  + 1;   MpAlarmXSet(DiagInterface.AlarmCore,'EventIDCode.2058');
		2060 :  AlarmCount[14 ] := AlarmCount[14]  + 1;   MpAlarmXSet(DiagInterface.AlarmCore,'EventIDCode.2060');
		2061 :  AlarmCount[15 ] := AlarmCount[15]  + 1;   MpAlarmXSet(DiagInterface.AlarmCore,'EventIDCode.2061');
		2063 :  AlarmCount[16 ] := AlarmCount[16]  + 1;   MpAlarmXSet(DiagInterface.AlarmCore,'EventIDCode.2063');
		2064 :  AlarmCount[17 ] := AlarmCount[17]  + 1;   MpAlarmXSet(DiagInterface.AlarmCore,'EventIDCode.2064');
		2066 :  AlarmCount[18 ] := AlarmCount[18]  + 1;   MpAlarmXSet(DiagInterface.AlarmCore,'EventIDCode.2066');
		2067 :  AlarmCount[19 ] := AlarmCount[19]  + 1;   MpAlarmXSet(DiagInterface.AlarmCore,'EventIDCode.2067');
		2068 :  AlarmCount[20 ] := AlarmCount[20]  + 1;   MpAlarmXSet(DiagInterface.AlarmCore,'EventIDCode.2068');
		2069 :  AlarmCount[21 ] := AlarmCount[21]  + 1;   MpAlarmXSet(DiagInterface.AlarmCore,'EventIDCode.2069');
		2070 :  AlarmCount[22 ] := AlarmCount[22]  + 1;   MpAlarmXSet(DiagInterface.AlarmCore,'EventIDCode.2070');
		2071 :  AlarmCount[23 ] := AlarmCount[23]  + 1;   MpAlarmXSet(DiagInterface.AlarmCore,'EventIDCode.2071');
		2074 :  AlarmCount[24 ] := AlarmCount[24]  + 1;   MpAlarmXSet(DiagInterface.AlarmCore,'EventIDCode.2074');
		2077 :  AlarmCount[25 ] := AlarmCount[25]  + 1;   MpAlarmXSet(DiagInterface.AlarmCore,'EventIDCode.2077');
		2080 :  AlarmCount[26 ] := AlarmCount[26]  + 1;   MpAlarmXSet(DiagInterface.AlarmCore,'EventIDCode.7392');
		2082 :  AlarmCount[27 ] := AlarmCount[27]  + 1;   MpAlarmXSet(DiagInterface.AlarmCore,'EventIDCode.2080');
		2083 :  AlarmCount[28 ] := AlarmCount[28]  + 1;   MpAlarmXSet(DiagInterface.AlarmCore,'EventIDCode.2083');
		2084 :  AlarmCount[29 ] := AlarmCount[29]  + 1;   MpAlarmXSet(DiagInterface.AlarmCore,'EventIDCode.2084');
		2085 :  AlarmCount[30 ] := AlarmCount[30]  + 1;   MpAlarmXSet(DiagInterface.AlarmCore,'EventIDCode.2085');
		2090 :  AlarmCount[31 ] := AlarmCount[31]  + 1;   MpAlarmXSet(DiagInterface.AlarmCore,'EventIDCode.2090');
		2091 :  AlarmCount[32 ] := AlarmCount[32]  + 1;   MpAlarmXSet(DiagInterface.AlarmCore,'EventIDCode.2091');
		2092 :  AlarmCount[33 ] := AlarmCount[33]  + 1;   MpAlarmXSet(DiagInterface.AlarmCore,'EventIDCode.2092');
		2093 :  AlarmCount[34 ] := AlarmCount[34]  + 1;   MpAlarmXSet(DiagInterface.AlarmCore,'EventIDCode.2093');
		2094 :  AlarmCount[35 ] := AlarmCount[35]  + 1;   MpAlarmXSet(DiagInterface.AlarmCore,'EventIDCode.2094');
		2095 :  AlarmCount[36 ] := AlarmCount[36]  + 1;   MpAlarmXSet(DiagInterface.AlarmCore,'EventIDCode.2095');
		2097 :  AlarmCount[37 ] := AlarmCount[37]  + 1;   MpAlarmXSet(DiagInterface.AlarmCore,'EventIDCode.2097');
		2098 :  AlarmCount[38 ] := AlarmCount[38]  + 1;   MpAlarmXSet(DiagInterface.AlarmCore,'EventIDCode.2098');
		2099 :  AlarmCount[39 ] := AlarmCount[39]  + 1;   MpAlarmXSet(DiagInterface.AlarmCore,'EventIDCode.2099');
		2100 :  AlarmCount[40 ] := AlarmCount[40]  + 1;   MpAlarmXSet(DiagInterface.AlarmCore,'EventIDCode.2100');
		2101 :  AlarmCount[41 ] := AlarmCount[41]  + 1;   MpAlarmXSet(DiagInterface.AlarmCore,'EventIDCode.2101');
		2102 :  AlarmCount[42 ] := AlarmCount[42]  + 1;   MpAlarmXSet(DiagInterface.AlarmCore,'EventIDCode.2102');
		2103 :  AlarmCount[43 ] := AlarmCount[43]  + 1;   MpAlarmXSet(DiagInterface.AlarmCore,'EventIDCode.2103');
		2104 :  AlarmCount[44 ] := AlarmCount[44]  + 1;   MpAlarmXSet(DiagInterface.AlarmCore,'EventIDCode.2104');
		2105 :  AlarmCount[45 ] := AlarmCount[45]  + 1;   MpAlarmXSet(DiagInterface.AlarmCore,'EventIDCode.2105');
		2106 :  AlarmCount[46 ] := AlarmCount[46]  + 1;   MpAlarmXSet(DiagInterface.AlarmCore,'EventIDCode.2106');
		2107 :  AlarmCount[47 ] := AlarmCount[47]  + 1;   MpAlarmXSet(DiagInterface.AlarmCore,'EventIDCode.2107');
		2108 :  AlarmCount[48 ] := AlarmCount[48]  + 1;   MpAlarmXSet(DiagInterface.AlarmCore,'EventIDCode.2108');
		2109 :  AlarmCount[49 ] := AlarmCount[49]  + 1;   MpAlarmXSet(DiagInterface.AlarmCore,'EventIDCode.2109');
		2110 :  AlarmCount[50 ] := AlarmCount[50]  + 1;   MpAlarmXSet(DiagInterface.AlarmCore,'EventIDCode.2110');
		2111 :  AlarmCount[51 ] := AlarmCount[51]  + 1;   MpAlarmXSet(DiagInterface.AlarmCore,'EventIDCode.2111');
		2112 :  AlarmCount[52 ] := AlarmCount[52]  + 1;   MpAlarmXSet(DiagInterface.AlarmCore,'EventIDCode.2112');
		4096 :  AlarmCount[53 ] := AlarmCount[53]  + 1;   MpAlarmXSet(DiagInterface.AlarmCore,'EventIDCode.4096');
		4097 :  AlarmCount[54 ] := AlarmCount[54]  + 1;   MpAlarmXSet(DiagInterface.AlarmCore,'EventIDCode.4097');
		4101 :  AlarmCount[55 ] := AlarmCount[55]  + 1;   MpAlarmXSet(DiagInterface.AlarmCore,'EventIDCode.4101');
		4102 :  AlarmCount[56 ] := AlarmCount[56]  + 1;   MpAlarmXSet(DiagInterface.AlarmCore,'EventIDCode.4102');
		6144 :  AlarmCount[57 ] := AlarmCount[57]  + 1;   MpAlarmXSet(DiagInterface.AlarmCore,'EventIDCode.6144');
		6165 :  AlarmCount[58 ] := AlarmCount[58]  + 1;   MpAlarmXSet(DiagInterface.AlarmCore,'EventIDCode.6165');
		6148 :  AlarmCount[59 ] := AlarmCount[59]  + 1;   MpAlarmXSet(DiagInterface.AlarmCore,'EventIDCode.6148');
		6149 :  AlarmCount[60 ] := AlarmCount[60]  + 1;   MpAlarmXSet(DiagInterface.AlarmCore,'EventIDCode.6149');
		6156 :  AlarmCount[61 ] := AlarmCount[61]  + 1;   MpAlarmXSet(DiagInterface.AlarmCore,'EventIDCode.6156');
		6157 :  AlarmCount[62 ] := AlarmCount[62]  + 1;   MpAlarmXSet(DiagInterface.AlarmCore,'EventIDCode.6157');
		6158 :  AlarmCount[63 ] := AlarmCount[63]  + 1;   MpAlarmXSet(DiagInterface.AlarmCore,'EventIDCode.6158');
		12288:  AlarmCount[64 ] := AlarmCount[64]  + 1;   MpAlarmXSet(DiagInterface.AlarmCore,'EventIDCode.12288');
		12291:  AlarmCount[65 ] := AlarmCount[65]  + 1;   MpAlarmXSet(DiagInterface.AlarmCore,'EventIDCode.12291');
		12293:  AlarmCount[66 ] := AlarmCount[66]  + 1;   MpAlarmXSet(DiagInterface.AlarmCore,'EventIDCode.12293');
		12294:  AlarmCount[67 ] := AlarmCount[67]  + 1;   MpAlarmXSet(DiagInterface.AlarmCore,'EventIDCode.12294');
		12295:  AlarmCount[68 ] := AlarmCount[68]  + 1;   MpAlarmXSet(DiagInterface.AlarmCore,'EventIDCode.12295');
		12296:  AlarmCount[69 ] := AlarmCount[69]  + 1;   MpAlarmXSet(DiagInterface.AlarmCore,'EventIDCode.12296');
		12297:  AlarmCount[70 ] := AlarmCount[70]  + 1;   MpAlarmXSet(DiagInterface.AlarmCore,'EventIDCode.12297');
		12298:  AlarmCount[71 ] := AlarmCount[71]  + 1;   MpAlarmXSet(DiagInterface.AlarmCore,'EventIDCode.12298');
		12299:  AlarmCount[72 ] := AlarmCount[72]  + 1;   MpAlarmXSet(DiagInterface.AlarmCore,'EventIDCode.12299');
		12300:  AlarmCount[73 ] := AlarmCount[73]  + 1;   MpAlarmXSet(DiagInterface.AlarmCore,'EventIDCode.12300');
		12301:  AlarmCount[74 ] := AlarmCount[74]  + 1;   MpAlarmXSet(DiagInterface.AlarmCore,'EventIDCode.12301');
		12302:  AlarmCount[75 ] := AlarmCount[75]  + 1;   MpAlarmXSet(DiagInterface.AlarmCore,'EventIDCode.12302');
		12303:  AlarmCount[76 ] := AlarmCount[76]  + 1;   MpAlarmXSet(DiagInterface.AlarmCore,'EventIDCode.12303');
		12304:  AlarmCount[77 ] := AlarmCount[77]  + 1;   MpAlarmXSet(DiagInterface.AlarmCore,'EventIDCode.12304');
		12305:  AlarmCount[78 ] := AlarmCount[78]  + 1;   MpAlarmXSet(DiagInterface.AlarmCore,'EventIDCode.12305');
		12307:  AlarmCount[79 ] := AlarmCount[79]  + 1;   MpAlarmXSet(DiagInterface.AlarmCore,'EventIDCode.12307');
		12312:  AlarmCount[80 ] := AlarmCount[80]  + 1;   MpAlarmXSet(DiagInterface.AlarmCore,'EventIDCode.12312');
		12313:  AlarmCount[81 ] := AlarmCount[81]  + 1;   MpAlarmXSet(DiagInterface.AlarmCore,'EventIDCode.12313');
		12314:  AlarmCount[82 ] := AlarmCount[82]  + 1;   MpAlarmXSet(DiagInterface.AlarmCore,'EventIDCode.12314');
		12315:  AlarmCount[83 ] := AlarmCount[83]  + 1;   MpAlarmXSet(DiagInterface.AlarmCore,'EventIDCode.12315');
		12316:  AlarmCount[84 ] := AlarmCount[84]  + 1;   MpAlarmXSet(DiagInterface.AlarmCore,'EventIDCode.12316');
		12317:  AlarmCount[85 ] := AlarmCount[85]  + 1;   MpAlarmXSet(DiagInterface.AlarmCore,'EventIDCode.12317');
		12320:  AlarmCount[86 ] := AlarmCount[86]  + 1;   MpAlarmXSet(DiagInterface.AlarmCore,'EventIDCode.12320');
		12322:  AlarmCount[87 ] := AlarmCount[87]  + 1;   MpAlarmXSet(DiagInterface.AlarmCore,'EventIDCode.12322');
		12323:  AlarmCount[88 ] := AlarmCount[88]  + 1;   MpAlarmXSet(DiagInterface.AlarmCore,'EventIDCode.12323');
		12328:  AlarmCount[89 ] := AlarmCount[89]  + 1;   MpAlarmXSet(DiagInterface.AlarmCore,'EventIDCode.12328');
		12330:  AlarmCount[90 ] := AlarmCount[90]  + 1;   MpAlarmXSet(DiagInterface.AlarmCore,'EventIDCode.12330');
		12331:  AlarmCount[91 ] := AlarmCount[91]  + 1;   MpAlarmXSet(DiagInterface.AlarmCore,'EventIDCode.12331');
		12333:  AlarmCount[92 ] := AlarmCount[92]  + 1;   MpAlarmXSet(DiagInterface.AlarmCore,'EventIDCode.12333');
		12334:  AlarmCount[93 ] := AlarmCount[93]  + 1;   MpAlarmXSet(DiagInterface.AlarmCore,'EventIDCode.12334');
		12335:  AlarmCount[94 ] := AlarmCount[94]  + 1;   MpAlarmXSet(DiagInterface.AlarmCore,'EventIDCode.12335');
		12336:  AlarmCount[95 ] := AlarmCount[95]  + 1;   MpAlarmXSet(DiagInterface.AlarmCore,'EventIDCode.12336');
		12337:  AlarmCount[96 ] := AlarmCount[96]  + 1;   MpAlarmXSet(DiagInterface.AlarmCore,'EventIDCode.12337');
		12338:  AlarmCount[97 ] := AlarmCount[97]  + 1;   MpAlarmXSet(DiagInterface.AlarmCore,'EventIDCode.12338');
		12340:  AlarmCount[98 ] := AlarmCount[98]  + 1;   MpAlarmXSet(DiagInterface.AlarmCore,'EventIDCode.12340');
		12341:  AlarmCount[99 ] := AlarmCount[99]  + 1;   MpAlarmXSet(DiagInterface.AlarmCore,'EventIDCode.12341');
		12342:  AlarmCount[100] := AlarmCount[100] + 1;   MpAlarmXSet(DiagInterface.AlarmCore,'EventIDCode.12342');
		12343:  AlarmCount[101] := AlarmCount[101] + 1;   MpAlarmXSet(DiagInterface.AlarmCore,'EventIDCode.12343');
		12344:  AlarmCount[102] := AlarmCount[102] + 1;   MpAlarmXSet(DiagInterface.AlarmCore,'EventIDCode.12344');
		12345:  AlarmCount[103] := AlarmCount[103] + 1;   MpAlarmXSet(DiagInterface.AlarmCore,'EventIDCode.12345');
		12346:  AlarmCount[104] := AlarmCount[104] + 1;   MpAlarmXSet(DiagInterface.AlarmCore,'EventIDCode.12346');
		12347:  AlarmCount[105] := AlarmCount[105] + 1;   MpAlarmXSet(DiagInterface.AlarmCore,'EventIDCode.12347');
		12348:  AlarmCount[106] := AlarmCount[106] + 1;   MpAlarmXSet(DiagInterface.AlarmCore,'EventIDCode.12348');
		4007:   AlarmCount[107] := AlarmCount[107] + 1;   MpAlarmXSet(DiagInterface.AlarmCore,'EventIDCode.4007');
		7230:   AlarmCount[108] := AlarmCount[108] + 1;   MpAlarmXSet(DiagInterface.AlarmCore,'EventIDCode.7230');
		4005:   AlarmCount[109] := AlarmCount[109] + 1;   MpAlarmXSet(DiagInterface.AlarmCore,'EventIDCode.4005');
		4098:   AlarmCount[110] := AlarmCount[110] + 1;   MpAlarmXSet(DiagInterface.AlarmCore,'EventIDCode.4098');
		9106:   AlarmCount[111] := AlarmCount[111] + 1;   MpAlarmXSet(DiagInterface.AlarmCore,'EventIDCode.9106');

		ELSE
			MpAlarmXSet(DiagInterface.AlarmCore,'EventIDCode.xxxx');
		END_CASE

END_ACTION
```

### Program Logical/Source/SampleTrak/Diagnostic/Logbook (IEC)
